Version 1	
*********************************************************************
Version Description:
- initial version
*********************************************************************
Version 2	
*********************************************************************
Version Description:
- Timeout control removed
- Assigning zero when It is not enabled, is removed.
*********************************************************************
*)


IF (C_Enable) THEN						(*Check if the functions is enabled*)
	fb_message(
	iCAN:= Obj_CAN, 
	iCanId:= X_MsgID, 
	iCanIdExtended:= S_Extended, 
	iTimeoutLimit:= Tm_MsgTmOut, 
	oByteCount=> , 
	oData=> , 
	oNewData=> , 
	oCanTimeout=> S_ER_TmOut, 
	oReceiverId=> , 
	oTooManyReceivers=> );	

	IF fb_message.oNewData THEN
	        
	   X_Byte_0 := fb_message.oData[0] ;
	   X_Byte_1 := fb_message.oData[1] ; 
	   X_Byte_2 := fb_message.oData[2] ; 
	   X_Byte_3 := fb_message.oData[3] ;
	   X_Byte_4 := fb_message.oData[4] ;
	   X_Byte_5 := fb_message.oData[5] ;
	   X_Byte_6 := fb_message.oData[6] ;
	   X_Byte_7 := fb_message.oData[7] ;  
	
	END_IF
	
END_IF


                  
END_FUNCTION_BLOCK

FUNCTION_BLOCK _FB_CanRx_Message_Unpack
  VAR_INPUT
    C_Enable : BOOL := FALSE;  (* Enable message *)
    Obj_CAN : POINTER TO tCan;  (* CAN Object derived from CAN_500_LIB *)
    X_MsgID : UDINT := 0;  (* Message ID *)
    Tm_MsgTmOut : TIME := TIME#500ms;  (* Message time limit *)
    S_Extended : BOOL := FALSE;  (* Message extended bit *)
  END_VAR
  VAR_OUTPUT
    S_ER_TmOut : BOOL;  (* Input data endpoints *)
    S_Bit_0 : BOOL;  (* Input data endpoints *)
    S_Bit_1 : BOOL;  (* Input data endpoints *)
    S_Bit_2 : BOOL;  (* Input data endpoints *)
    S_Bit_3 : BOOL;  (* Input data endpoints *)
    S_Bit_4 : BOOL;  (* Input data endpoints *)
    S_Bit_5 : BOOL;  (* Input data endpoints *)
    S_Bit_6 : BOOL;  (* Input data endpoints *)
    S_Bit_7 : BOOL;  (* Input data endpoints *)
    X_Byte_0 : BYTE;  (* Input data endpoints *)
    S_Bit_8 : BOOL;  (* Input data endpoints *)
    S_Bit_9 : BOOL;  (* Input data endpoints *)
    S_Bit_10 : BOOL;  (* Input data endpoints *)
    S_Bit_11 : BOOL;  (* Input data endpoints *)
    S_Bit_12 : BOOL;  (* Input data endpoints *)
    S_Bit_13 : BOOL;  (* Input data endpoints *)
    S_Bit_14 : BOOL;  (* Input data endpoints *)
    S_Bit_15 : BOOL;  (* Input data endpoints *)
    X_Byte_1 : BYTE;  (* Input data endpoints *)
    X_Word_0 : WORD;  (* Input data endpoints *)
    S_Bit_16 : BOOL;  (* Input data endpoints *)
    S_Bit_17 : BOOL;  (* Input data endpoints *)
    S_Bit_18 : BOOL;  (* Input data endpoints *)
    S_Bit_19 : BOOL;  (* Input data endpoints *)
    S_Bit_20 : BOOL;  (* Input data endpoints *)
    S_Bit_21 : BOOL;  (* Input data endpoints *)
    S_Bit_22 : BOOL;  (* Input data endpoints *)
    S_Bit_23 : BOOL;  (* Input data endpoints *)
    X_Byte_2 : BYTE;  (* Input data endpoints *)
    S_Bit_24 : BOOL;  (* Input data endpoints *)
    S_Bit_25 : BOOL;  (* Input data endpoints *)
    S_Bit_26 : BOOL;  (* Input data endpoints *)
    S_Bit_27 : BOOL;  (* Input data endpoints *)
    S_Bit_28 : BOOL;  (* Input data endpoints *)
    S_Bit_29 : BOOL;  (* Input data endpoints *)
    S_Bit_30 : BOOL;  (* Input data endpoints *)
    S_Bit_31 : BOOL;  (* Input data endpoints *)
    X_Byte_3 : BYTE;  (* Input data endpoints *)
    S_Bit_32 : BOOL;  (* Input data endpoints *)
    S_Bit_33 : BOOL;  (* Input data endpoints *)
    S_Bit_34 : BOOL;  (* Input data endpoints *)
    S_Bit_35 : BOOL;  (* Input data endpoints *)
    S_Bit_36 : BOOL;  (* Input data endpoints *)
    S_Bit_37 : BOOL;  (* Input data endpoints *)
    S_Bit_38 : BOOL;  (* Input data endpoints *)
    S_Bit_39 : BOOL;  (* Input data endpoints *)
    X_Byte_4 : BYTE;  (* Input data endpoints *)
    S_Bit_40 : BOOL;  (* Input data endpoints *)
    S_Bit_41 : BOOL;  (* Input data endpoints *)
    S_Bit_42 : BOOL;  (* Input data endpoints *)
    S_Bit_43 : BOOL;  (* Input data endpoints *)
    S_Bit_44 : BOOL;  (* Input data endpoints *)
    S_Bit_45 : BOOL;  (* Input data endpoints *)
    S_Bit_46 : BOOL;  (* Input data endpoints *)
    S_Bit_47 : BOOL;  (* Input data endpoints *)
    X_Byte_5 : BYTE;  (* Input data endpoints *)
    X_Word_2 : WORD;  (* Input data endpoints *)
    S_Bit_48 : BOOL;  (* Input data endpoints *)
    S_Bit_49 : BOOL;  (* Input data endpoints *)
    S_Bit_50 : BOOL;  (* Input data endpoints *)
    S_Bit_51 : BOOL;  (* Input data endpoints *)
    S_Bit_52 : BOOL;  (* Input data endpoints *)
    S_Bit_53 : BOOL;  (* Input data endpoints *)
    S_Bit_54 : BOOL;  (* Input data endpoints *)
    S_Bit_55 : BOOL;  (* Input data endpoints *)
    X_Byte_6 : BYTE;  (* Input data endpoints *)
    S_Bit_56 : BOOL;  (* Input data endpoints *)
    S_Bit_57 : BOOL;  (* Input data endpoints *)
    S_Bit_58 : BOOL;  (* Input data endpoints *)
    S_Bit_59 : BOOL;  (* Input data endpoints *)
    S_Bit_60 : BOOL;  (* Input data endpoints *)
    S_Bit_61 : BOOL;  (* Input data endpoints *)
    S_Bit_62 : BOOL;  (* Input data endpoints *)
    S_Bit_63 : BOOL;  (* Input data endpoints *)
    X_Byte_7 : BYTE;  (* Input data endpoints *)
  END_VAR
  VAR
    fb_message : CanRx;  (* Library object container *)
    STIMEOUT : BOOL;
  END_VAR

                    (*
**********************************************************************
Bozankaya A.Ş.
**********************************************************************
Name					: _FB_CanRx_Message
POU Type				: FB
Created by 				: E.TURKER , BZK.
Creation Date 			: 09-03-2022
Modifications			: see version description below


FB Description:
This FB handles the RX can messages according to CAN_500_LIB
*********************************************************************

Version 1	
*********************************************************************
Version Description:
- initial version
*********************************************************************
Version 2	
*********************************************************************
Version Description:
- Word and dword transitions are removed
*********************************************************************
*)


IF (C_Enable) THEN				(*Check if the function is enabled*)
	fb_message(
	iCAN:= Obj_CAN, 
	iCanId:= X_MsgID, 
	iCanIdExtended:= S_Extended, 
	iTimeoutLimit:= Tm_MsgTmOut, 
	oByteCount=> , 
	oData=> , 
	oNewData=> , 
	oCanTimeout=> S_ER_TmOut, 
	oReceiverId=> , 
	oTooManyReceivers=> );
	
	
	
	IF fb_message.oNewData THEN			(*Check if the new message is received*)

			X_Byte_0 := fb_message.oData[0] ;
			X_Byte_1 := fb_message.oData[1] ; 
			X_Byte_2 := fb_message.oData[2] ; 
			X_Byte_3 := fb_message.oData[3] ;
			X_Byte_4 := fb_message.oData[4] ;
			X_Byte_5 := fb_message.oData[5] ;
			X_Byte_6 := fb_message.oData[6] ;
			X_Byte_7 := fb_message.oData[7] ;  
			
	END_IF
   
	
	
ELSE	
	
			X_Byte_0 := 0 ;
			X_Byte_1 := 0 ;
			X_Byte_2 := 0 ;
			X_Byte_3 := 0 ;
			X_Byte_4 := 0 ;
			X_Byte_5 := 0 ;
			X_Byte_6 := 0 ;
			X_Byte_7 := 0 ;
			
END_IF

			S_Bit_0  := BYTE_TO_BOOL(X_Byte_0 AND 2#00000001);
			S_Bit_1  := BYTE_TO_BOOL(X_Byte_0 AND 2#00000010);
			S_Bit_2  := BYTE_TO_BOOL(X_Byte_0 AND 2#00000100);
			S_Bit_3  := BYTE_TO_BOOL(X_Byte_0 AND 2#00001000);
			S_Bit_4  := BYTE_TO_BOOL(X_Byte_0 AND 2#00010000);
			S_Bit_5  := BYTE_TO_BOOL(X_Byte_0 AND 2#00100000);
			S_Bit_6  := BYTE_TO_BOOL(X_Byte_0 AND 2#01000000);
			S_Bit_7  := BYTE_TO_BOOL(X_Byte_0 AND 2#10000000);
			S_Bit_8  := BYTE_TO_BOOL(X_Byte_1 AND 2#00000001);
			S_Bit_9  := BYTE_TO_BOOL(X_Byte_1 AND 2#00000010);
			S_Bit_10  := BYTE_TO_BOOL(X_Byte_1 AND 2#00000100);
			S_Bit_11  := BYTE_TO_BOOL(X_Byte_1 AND 2#00001000);
			S_Bit_12  := BYTE_TO_BOOL(X_Byte_1 AND 2#00010000);
			S_Bit_13  := BYTE_TO_BOOL(X_Byte_1 AND 2#00100000);
			S_Bit_14  := BYTE_TO_BOOL(X_Byte_1 AND 2#01000000);
			S_Bit_15  := BYTE_TO_BOOL(X_Byte_1 AND 2#10000000);
			S_Bit_16  := BYTE_TO_BOOL(X_Byte_2 AND 2#00000001);
			S_Bit_17  := BYTE_TO_BOOL(X_Byte_2 AND 2#00000010);
			S_Bit_18  := BYTE_TO_BOOL(X_Byte_2 AND 2#00000100);
			S_Bit_19  := BYTE_TO_BOOL(X_Byte_2 AND 2#00001000);
			S_Bit_20  := BYTE_TO_BOOL(X_Byte_2 AND 2#00010000);
			S_Bit_21  := BYTE_TO_BOOL(X_Byte_2 AND 2#00100000);
			S_Bit_22  := BYTE_TO_BOOL(X_Byte_2 AND 2#01000000);
			S_Bit_23  := BYTE_TO_BOOL(X_Byte_2 AND 2#10000000);
			S_Bit_24  := BYTE_TO_BOOL(X_Byte_3 AND 2#00000001);
			S_Bit_25  := BYTE_TO_BOOL(X_Byte_3 AND 2#00000010);
			S_Bit_26  := BYTE_TO_BOOL(X_Byte_3 AND 2#00000100);
			S_Bit_27  := BYTE_TO_BOOL(X_Byte_3 AND 2#00001000);
			S_Bit_28  := BYTE_TO_BOOL(X_Byte_3 AND 2#00010000);
			S_Bit_29  := BYTE_TO_BOOL(X_Byte_3 AND 2#00100000);
			S_Bit_30  := BYTE_TO_BOOL(X_Byte_3 AND 2#01000000);
			S_Bit_31  := BYTE_TO_BOOL(X_Byte_3 AND 2#10000000);
			S_Bit_32  := BYTE_TO_BOOL(X_Byte_4 AND 2#00000001);
			S_Bit_33  := BYTE_TO_BOOL(X_Byte_4 AND 2#00000010);
			S_Bit_34  := BYTE_TO_BOOL(X_Byte_4 AND 2#00000100);
			S_Bit_35  := BYTE_TO_BOOL(X_Byte_4 AND 2#00001000);
			S_Bit_36  := BYTE_TO_BOOL(X_Byte_4 AND 2#00010000);
			S_Bit_37  := BYTE_TO_BOOL(X_Byte_4 AND 2#00100000);
			S_Bit_38  := BYTE_TO_BOOL(X_Byte_4 AND 2#01000000);
			S_Bit_39  := BYTE_TO_BOOL(X_Byte_4 AND 2#10000000);
			S_Bit_40  := BYTE_TO_BOOL(X_Byte_5 AND 2#00000001);
			S_Bit_41  := BYTE_TO_BOOL(X_Byte_5 AND 2#00000010);
			S_Bit_42  := BYTE_TO_BOOL(X_Byte_5 AND 2#00000100);
			S_Bit_43  := BYTE_TO_BOOL(X_Byte_5 AND 2#00001000);
			S_Bit_44  := BYTE_TO_BOOL(X_Byte_5 AND 2#00010000);
			S_Bit_45  := BYTE_TO_BOOL(X_Byte_5 AND 2#00100000);
			S_Bit_46  := BYTE_TO_BOOL(X_Byte_5 AND 2#01000000);
			S_Bit_47  := BYTE_TO_BOOL(X_Byte_5 AND 2#10000000);
			S_Bit_48  := BYTE_TO_BOOL(X_Byte_6 AND 2#00000001);
			S_Bit_49  := BYTE_TO_BOOL(X_Byte_6 AND 2#00000010);
			S_Bit_50  := BYTE_TO_BOOL(X_Byte_6 AND 2#00000100);
			S_Bit_51  := BYTE_TO_BOOL(X_Byte_6 AND 2#00001000);
			S_Bit_52  := BYTE_TO_BOOL(X_Byte_6 AND 2#00010000);
			S_Bit_53  := BYTE_TO_BOOL(X_Byte_6 AND 2#00100000);
			S_Bit_54  := BYTE_TO_BOOL(X_Byte_6 AND 2#01000000);
			S_Bit_55  := BYTE_TO_BOOL(X_Byte_6 AND 2#10000000);
			S_Bit_56  := BYTE_TO_BOOL(X_Byte_7 AND 2#00000001);
			S_Bit_57  := BYTE_TO_BOOL(X_Byte_7 AND 2#00000010);
			S_Bit_58  := BYTE_TO_BOOL(X_Byte_7 AND 2#00000100);
			S_Bit_59  := BYTE_TO_BOOL(X_Byte_7 AND 2#00001000);
			S_Bit_60  := BYTE_TO_BOOL(X_Byte_7 AND 2#00010000);
			S_Bit_61  := BYTE_TO_BOOL(X_Byte_7 AND 2#00100000);
			S_Bit_62  := BYTE_TO_BOOL(X_Byte_7 AND 2#01000000);
			S_Bit_63  := BYTE_TO_BOOL(X_Byte_7 AND 2#10000000);

                  
END_FUNCTION_BLOCK

FUNCTION_BLOCK _FB_CanTx_Message
  VAR_INPUT
    C_Enable : BOOL := FALSE;  (* Enable message *)
    Obj_CAN : POINTER TO tCan;  (* CAN Object derived from CAN_500_LIB *)
    X_MsgID : UDINT := 0;  (* Message ID *)
    Tm_CycleTime : TIME := TIME#500ms;  (* Message time limit *)
    N_Msg_Dlc : BYTE := 8;  (* Message dlc *)
    S_Extended : BOOL := FALSE;  (* Message extended bit *)
    X_Byte_0 : BYTE := 16#FF;  (* Message Datas *)
    X_Byte_1 : BYTE := 16#FF;  (* Message Datas *)
    X_Byte_2 : BYTE := 16#FF;  (* Message Datas *)
    X_Byte_3 : BYTE := 16#FF;  (* Message Datas *)
    X_Byte_4 : BYTE := 16#FF;  (* Message Datas *)
    X_Byte_5 : BYTE := 16#FF;  (* Message Datas *)
    X_Byte_6 : BYTE := 16#FF;  (* Message Datas *)
    X_Byte_7 : BYTE := 16#FF;  (* Message Datas *)
  END_VAR
  VAR_OUTPUT
    S_Sent_Ok : BOOL;  (* Data sent acknowledge *)
  END_VAR
  VAR
    fb_message : CanTx;  (* Library object container *)
    Arr_X_Data : ARRAY[0..7] OF BYTE;  (* Message data array *)
  END_VAR

                    (*
**********************************************************************
Bozankaya A.Ş.
**********************************************************************
Name					: _FB_CanTx_Message
POU Type				: FB
Created by 				: E.TURKER , BZK.
Creation Date 			: 09-03-2022
Modifications			: see version description below


FB Description:
This FB handles the TX can messages according to CAN_500_LIB
*********************************************************************

Version 1	
*********************************************************************
Version Description:
- initial version
*********************************************************************
Version 2	
*********************************************************************
Version Description:
- Assigning zero when It is not enabled, is removed.
*********************************************************************
*)

IF C_Enable THEN				(*Check if the function is enabled*)
			
			Arr_X_Data [0] := X_Byte_0;
			Arr_X_Data [1] := X_Byte_1;
			Arr_X_Data [2] := X_Byte_2;
			Arr_X_Data [3] := X_Byte_3;
			Arr_X_Data [4] := X_Byte_4;
			Arr_X_Data [5] := X_Byte_5;		
            Arr_X_Data [6] := X_Byte_6;
			Arr_X_Data [7] := X_Byte_7;

END_IF

fb_message(
	
	iEnable:= C_Enable, 
	iCAN:= Obj_CAN, 
	iForceSend:= FALSE, 
	iTransmitRate:= Tm_CycleTime, 
	iCanId:= X_MsgID, 
	iCanIdExtended:= S_Extended, 
	iByteCount:= N_Msg_Dlc, 
	iData:= Arr_X_Data, 
	oTransmitterId=> , 
	oTooManyTransmitters=> , 
	oMsgSent=> S_Sent_Ok );
	
                  
END_FUNCTION_BLOCK

FUNCTION_BLOCK _FB_CanTx_Message_Unpack
  VAR_INPUT
    C_Enable : BOOL := FALSE;  (* Enable message *)
    Obj_CAN : POINTER TO tCan;  (* CAN Object derived from CAN_500_LIB *)
    X_MsgID : UDINT := 0;  (* Message ID *)
    Tm_CycleTime : TIME := TIME#500ms;  (* Message time limit *)
    S_Extended : BOOL := FALSE;  (* Message extended bit *)
    N_Msg_Dlc : BYTE;
    S_Bit_0 : BOOL := FALSE;  (* Message Datas *)
    S_Bit_1 : BOOL := FALSE;  (* Message Datas *)
    S_Bit_2 : BOOL := FALSE;  (* Message Datas *)
    S_Bit_3 : BOOL := FALSE;  (* Message Datas *)
    S_Bit_4 : BOOL := FALSE;  (* Message Datas *)
    S_Bit_5 : BOOL := FALSE;  (* Message Datas *)
    S_Bit_6 : BOOL := FALSE;  (* Message Datas *)
    S_Bit_7 : BOOL := FALSE;  (* Message Datas *)
    X_Byte_0 : BYTE := 16#0;  (* Message Datas *)
    S_Bit_8 : BOOL := FALSE;  (* Message Datas *)
    S_Bit_9 : BOOL := FALSE;  (* Message Datas *)
    S_Bit_10 : BOOL := FALSE;  (* Message Datas *)
    S_Bit_11 : BOOL := FALSE;  (* Message Datas *)
    S_Bit_12 : BOOL := FALSE;  (* Message Datas *)
    S_Bit_13 : BOOL := FALSE;  (* Message Datas *)
    S_Bit_14 : BOOL := FALSE;  (* Message Datas *)
    S_Bit_15 : BOOL := FALSE;  (* Message Datas *)
    X_Byte_1 : BYTE := 16#0;  (* Message Datas *)
    S_Bit_16 : BOOL := FALSE;  (* Message Datas *)
    S_Bit_17 : BOOL := FALSE;  (* Message Datas *)
    S_Bit_18 : BOOL := FALSE;  (* Message Datas *)
    S_Bit_19 : BOOL := FALSE;  (* Message Datas *)
    S_Bit_20 : BOOL := FALSE;  (* Message Datas *)
    S_Bit_21 : BOOL := FALSE;  (* Message Datas *)
    S_Bit_22 : BOOL := FALSE;  (* Message Datas *)
    S_Bit_23 : BOOL := FALSE;  (* Message Datas *)
    X_Byte_2 : BYTE := 16#0;  (* Message Datas *)
    S_Bit_24 : BOOL := FALSE;  (* Message Datas *)
    S_Bit_25 : BOOL := FALSE;  (* Message Datas *)
    S_Bit_26 : BOOL := FALSE;  (* Message Datas *)
    S_Bit_27 : BOOL := FALSE;  (* Message Datas *)
    S_Bit_28 : BOOL := FALSE;  (* Message Datas *)
    S_Bit_29 : BOOL := FALSE;  (* Message Datas *)
    S_Bit_30 : BOOL := FALSE;  (* Message Datas *)
    S_Bit_31 : BOOL := FALSE;  (* Message Datas *)
    X_Byte_3 : BYTE := 16#0;  (* Message Datas *)
    S_Bit_32 : BOOL := FALSE;  (* Message Datas *)
    S_Bit_33 : BOOL := FALSE;  (* Message Datas *)
    S_Bit_34 : BOOL := FALSE;  (* Message Datas *)
    S_Bit_35 : BOOL := FALSE;  (* Message Datas *)
    S_Bit_36 : BOOL := FALSE;  (* Message Datas *)
    S_Bit_37 : BOOL := FALSE;  (* Message Datas *)
    S_Bit_38 : BOOL := FALSE;  (* Message Datas *)
    S_Bit_39 : BOOL := FALSE;  (* Message Datas *)
    X_Byte_4 : BYTE := 16#0;  (* Message Datas *)
    S_Bit_40 : BOOL := FALSE;  (* Message Datas *)
    S_Bit_41 : BOOL := FALSE;  (* Message Datas *)
    S_Bit_42 : BOOL := FALSE;  (* Message Datas *)
    S_Bit_43 : BOOL := FALSE;  (* Message Datas *)
    S_Bit_44 : BOOL := FALSE;  (* Message Datas *)
    S_Bit_45 : BOOL := FALSE;  (* Message Datas *)
    S_Bit_46 : BOOL := FALSE;  (* Message Datas *)
    S_Bit_47 : BOOL := FALSE;  (* Message Datas *)
    X_Byte_5 : BYTE := 16#0;  (* Message Datas *)
    S_Bit_48 : BOOL := FALSE;  (* Message Datas *)
    S_Bit_49 : BOOL := FALSE;  (* Message Datas *)
    S_Bit_50 : BOOL := FALSE;  (* Message Datas *)
    S_Bit_51 : BOOL := FALSE;  (* Message Datas *)
    S_Bit_52 : BOOL := FALSE;  (* Message Datas *)
    S_Bit_53 : BOOL := FALSE;  (* Message Datas *)
    S_Bit_54 : BOOL := FALSE;  (* Message Datas *)
    S_Bit_55 : BOOL := FALSE;  (* Message Datas *)
    X_Byte_6 : BYTE := 16#0;  (* Message Datas *)
    S_Bit_56 : BOOL := FALSE;  (* Message Datas *)
    S_Bit_57 : BOOL := FALSE;  (* Message Datas *)
    S_Bit_58 : BOOL := FALSE;  (* Message Datas *)
    S_Bit_59 : BOOL := FALSE;  (* Message Datas *)
    S_Bit_60 : BOOL := FALSE;  (* Message Datas *)
    S_Bit_61 : BOOL := FALSE;  (* Message Datas *)
    S_Bit_62 : BOOL := FALSE;  (* Message Datas *)
    S_Bit_63 : BOOL := FALSE;  (* Message Datas *)
    X_Byte_7 : BYTE := 16#0;  (* Message Datas *)
  END_VAR
  VAR_OUTPUT
    S_Sent_Ok : BOOL;  (* Data sent acknowledge *)
  END_VAR
  VAR
    fb_message : CanTx;  (* Library object container *)
    DATA : ARRAY[0..7] OF BYTE;  (* Message data array *)
    _FB_Pack_Bit_To_Byte_01 : _FB_PACK_8BITS_TO_BYTE;
    _FB_Pack_Bit_To_Byte_02 : _FB_PACK_8BITS_TO_BYTE;
    _FB_Pack_Bit_To_Byte_03 : _FB_PACK_8BITS_TO_BYTE;
    _FB_Pack_Bit_To_Byte_04 : _FB_PACK_8BITS_TO_BYTE;
    _FB_Pack_Bit_To_Byte_05 : _FB_PACK_8BITS_TO_BYTE;
    _FB_Pack_Bit_To_Byte_06 : _FB_PACK_8BITS_TO_BYTE;
    _FB_Pack_Bit_To_Byte_07 : _FB_PACK_8BITS_TO_BYTE;
    _FB_Pack_Bit_To_Byte_08 : _FB_PACK_8BITS_TO_BYTE;
  END_VAR

                    (*
**********************************************************************
Bozankaya A.Ş.
**********************************************************************
Name					: _FB_CanTx_Message
POU Type				: FB
Created by 				: E.TURKER , BZK.
Creation Date 			: 09-03-2022
Modifications			: see version description below


FB Description:
This FB handles the TX can messages according to CAN_500_LIB
*********************************************************************

Version 1	
*********************************************************************
Version Description:
- initial version
*********************************************************************
Version 1	
*********************************************************************
Version Description:
- WORD and DWORD transitions are removed
*********************************************************************
*)

IF X_Byte_0 <> 0 THEN
	
	DATA [0] := X_Byte_0;
	
ELSIF S_Bit_0 OR S_Bit_1 OR S_Bit_2 OR S_Bit_3 OR S_Bit_4 OR S_Bit_5 OR S_Bit_6 OR S_Bit_7 THEN			(*Check the bits, pack and assign to the output data*)
	_FB_Pack_Bit_To_Byte_01(
	S_Bit_0:= S_Bit_0, 
	S_Bit_1:= S_Bit_1, 
	S_Bit_2:= S_Bit_2, 
	S_Bit_3:= S_Bit_3, 
	S_Bit_4:= S_Bit_4, 
	S_Bit_5:= S_Bit_5, 
	S_Bit_6:= S_Bit_6, 
	S_Bit_7:= S_Bit_7, 
	X_Byte_0=> DATA [0]);
ELSE
	DATA [0] := 0;
END_IF
		
IF X_Byte_1 <> 0 THEN
	DATA [1] := X_Byte_1;
ELSIF S_Bit_8 OR S_Bit_9 OR S_Bit_10 OR S_Bit_11 OR S_Bit_12 OR S_Bit_13 OR S_Bit_14 OR S_Bit_15 THEN			(*Check the bits, pack and assign to the output data*)
	_FB_Pack_Bit_To_Byte_02(
	S_Bit_0:= S_Bit_8, 
	S_Bit_1:= S_Bit_9, 
	S_Bit_2:= S_Bit_10, 
	S_Bit_3:= S_Bit_11, 
	S_Bit_4:= S_Bit_12, 
	S_Bit_5:= S_Bit_13, 
	S_Bit_6:= S_Bit_14, 
	S_Bit_7:= S_Bit_15, 
	X_Byte_0=> DATA [1]);
ELSE
	DATA [1] :=0;
END_IF
	

IF X_Byte_2 <> 0 THEN
	DATA [2] := X_Byte_2;
ELSIF S_Bit_16 OR S_Bit_17 OR S_Bit_18 OR S_Bit_19 OR S_Bit_20 OR S_Bit_21 OR S_Bit_22 OR S_Bit_23 THEN				(*Check the bits, pack and assign to the output data*)
	_FB_Pack_Bit_To_Byte_03(
	S_Bit_0:= S_Bit_16, 
	S_Bit_1:= S_Bit_17, 
	S_Bit_2:= S_Bit_18, 
	S_Bit_3:= S_Bit_19, 
	S_Bit_4:= S_Bit_20, 
	S_Bit_5:= S_Bit_21, 
	S_Bit_6:= S_Bit_22, 
	S_Bit_7:= S_Bit_23, 
	X_Byte_0=> DATA [2]);
ELSE
	DATA [2] :=0;
END_IF
		
IF X_Byte_3 <> 0 THEN
	DATA [3] := X_Byte_3;
ELSIF S_Bit_24 OR S_Bit_25 OR S_Bit_26 OR S_Bit_27 OR S_Bit_28 OR S_Bit_29 OR S_Bit_30 OR S_Bit_31 THEN				(*Check the bits, pack and assign to the output data*)
	_FB_Pack_Bit_To_Byte_04(
	S_Bit_0:= S_Bit_24, 
	S_Bit_1:= S_Bit_25, 
	S_Bit_2:= S_Bit_26, 
	S_Bit_3:= S_Bit_27, 
	S_Bit_4:= S_Bit_28, 
	S_Bit_5:= S_Bit_29, 
	S_Bit_6:= S_Bit_30, 
	S_Bit_7:= S_Bit_31, 
	X_Byte_0=> DATA [3]);
ELSE
	DATA [3] :=0;
END_IF



IF X_Byte_4 <> 0 THEN
	DATA [4] := X_Byte_4;
ELSIF S_Bit_32 OR S_Bit_33 OR S_Bit_34 OR S_Bit_35 OR S_Bit_36 OR S_Bit_37 OR S_Bit_38 OR S_Bit_39 THEN				(*Check the bits, pack and assign to the output data*)
	_FB_Pack_Bit_To_Byte_05(
	S_Bit_0:= S_Bit_32, 
	S_Bit_1:= S_Bit_33, 
	S_Bit_2:= S_Bit_34, 
	S_Bit_3:= S_Bit_35, 
	S_Bit_4:= S_Bit_36, 
	S_Bit_5:= S_Bit_37, 
	S_Bit_6:= S_Bit_38, 
	S_Bit_7:= S_Bit_39, 
	X_Byte_0=> DATA [4]);	
ELSE
	DATA [4] :=0;
END_IF
		
IF X_Byte_5 <> 0 THEN
	DATA [5] := X_Byte_5;
ELSIF S_Bit_40 OR S_Bit_41 OR S_Bit_42 OR S_Bit_43 OR S_Bit_44 OR S_Bit_45 OR S_Bit_46 OR S_Bit_47 THEN				(*Check the bits, pack and assign to the output data*)
	_FB_Pack_Bit_To_Byte_06(
	S_Bit_0:= S_Bit_40, 
	S_Bit_1:= S_Bit_41, 
	S_Bit_2:= S_Bit_42, 
	S_Bit_3:= S_Bit_43, 
	S_Bit_4:= S_Bit_44, 
	S_Bit_5:= S_Bit_45, 
	S_Bit_6:= S_Bit_46, 
	S_Bit_7:= S_Bit_47, 
	X_Byte_0=> DATA [5]);
ELSE
	DATA [5] :=0;
END_IF

	

IF X_Byte_6 <> 0 THEN
	DATA [6] := X_Byte_6;
ELSIF S_Bit_48 OR S_Bit_49 OR S_Bit_50 OR S_Bit_51 OR S_Bit_52 OR S_Bit_53 OR S_Bit_54 OR S_Bit_55 THEN				(*Check the bits, pack and assign to the output data*)
	_FB_Pack_Bit_To_Byte_07(
	S_Bit_0:= S_Bit_48, 
	S_Bit_1:= S_Bit_49, 
	S_Bit_2:= S_Bit_50, 
	S_Bit_3:= S_Bit_51, 
	S_Bit_4:= S_Bit_52, 
	S_Bit_5:= S_Bit_53, 
	S_Bit_6:= S_Bit_54, 
	S_Bit_7:= S_Bit_55, 
	X_Byte_0=> DATA [6]);
ELSE
	DATA [6] :=0;
END_IF
		
IF X_Byte_7 <> 0 THEN
	DATA [7] := X_Byte_7;
ELSIF S_Bit_56 OR S_Bit_57 OR S_Bit_58 OR S_Bit_59 OR S_Bit_60 OR S_Bit_61 OR S_Bit_62 OR S_Bit_63 THEN				(*Check the bits, pack and assign to the output data*)
	_FB_Pack_Bit_To_Byte_08(
	S_Bit_0:= S_Bit_56, 
	S_Bit_1:= S_Bit_57, 
	S_Bit_2:= S_Bit_58, 
	S_Bit_3:= S_Bit_59, 
	S_Bit_4:= S_Bit_60, 
	S_Bit_5:= S_Bit_61, 
	S_Bit_6:= S_Bit_62, 
	S_Bit_7:= S_Bit_63, 
	X_Byte_0=> DATA [7]);
ELSE
	DATA [7] :=0;
END_IF


fb_message(
	iEnable:= C_Enable, 
	iCAN:= Obj_CAN, 
	iForceSend:= FALSE, 
	iTransmitRate:= Tm_CycleTime, 
	iCanId:= X_MsgID, 
	iCanIdExtended:= S_Extended, 
	iByteCount:= N_Msg_Dlc, 
	iData:= DATA, 
	oTransmitterId=> , 
	oTooManyTransmitters=> , 
	oMsgSent=> S_Sent_Ok );
                  
END_FUNCTION_BLOCK

FUNCTION_BLOCK _FB_LfMon
  VAR_INPUT
    X_Lf : UINT;
    P_Lf_Timeout : TIME;
  END_VAR
  VAR_OUTPUT
    S_Lf_Timeout : BOOL;
  END_VAR
  VAR
    X_Lf_Old : UINT;
    TON_0 : TON;
  END_VAR

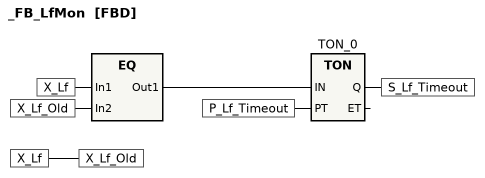
(* FBD diagram, written out as Structured Text *)
TON_0(IN := X_Lf = X_Lf_Old, PT := P_Lf_Timeout);
S_Lf_Timeout := TON_0.Q;
X_Lf_Old := X_Lf;
END_FUNCTION_BLOCK

FUNCTION_BLOCK _FB_PACK_8BITS_TO_BYTE
  VAR_INPUT
    S_BIT_0 : BOOL;  (* Less significant part *)
    S_BIT_1 : BOOL;
    S_BIT_2 : BOOL;
    S_BIT_3 : BOOL;
    S_BIT_4 : BOOL;
    S_BIT_5 : BOOL;
    S_BIT_6 : BOOL;
    S_BIT_7 : BOOL;  (* Most significant part *)
  END_VAR
  VAR_OUTPUT
    X_BYTE_0 : BYTE;  (* Output data *)
  END_VAR
  VAR
    X_Cont_Byte : BYTE;  (* Container data for shifting operation *)
  END_VAR

                    X_Cont_Byte 	:= BOOL_TO_BYTE(S_BIT_7) OR X_Cont_Byte;			
X_Cont_Byte		:= SHL(X_Cont_Byte, 1);
X_Cont_Byte     := BOOL_TO_BYTE(S_BIT_6) OR X_Cont_Byte;
X_Cont_Byte		:= SHL(X_Cont_Byte, 1);
X_Cont_Byte     := BOOL_TO_BYTE(S_BIT_5) OR X_Cont_Byte;
X_Cont_Byte		:= SHL(X_Cont_Byte, 1);
X_Cont_Byte     := BOOL_TO_BYTE(S_BIT_4) OR X_Cont_Byte;
X_Cont_Byte		:= SHL(X_Cont_Byte, 1);
X_Cont_Byte     := BOOL_TO_BYTE(S_BIT_3) OR X_Cont_Byte;
X_Cont_Byte		:= SHL(X_Cont_Byte, 1);
X_Cont_Byte     := BOOL_TO_BYTE(S_BIT_2) OR X_Cont_Byte;
X_Cont_Byte		:= SHL(X_Cont_Byte, 1);
X_Cont_Byte     := BOOL_TO_BYTE(S_BIT_1) OR X_Cont_Byte;
X_Cont_Byte		:= SHL(X_Cont_Byte, 1);
X_Cont_Byte     := BOOL_TO_BYTE(S_BIT_0) OR X_Cont_Byte;
X_BYTE_0		:= X_Cont_Byte;
X_Cont_Byte		:=0;
                  
END_FUNCTION_BLOCK

FUNCTION_BLOCK _FB_PACK_BYTE_TO_DINT
  VAR_INPUT
    X_Byte_0 : BYTE;  (* Input less significant part *)
    X_Byte_1 : BYTE;
    X_Byte_2 : BYTE;
    X_Byte_3 : BYTE;
    X_Byte_4 : BYTE;
    X_Byte_5 : BYTE;
    X_Byte_6 : BYTE;
    X_Byte_7 : BYTE;  (* Input most significant part *)
  END_VAR
  VAR_OUTPUT
    X_Dint_0 : DINT;
  END_VAR
  VAR
    X_Cont_Udint : UDINT;  (* Container data for shifting operation *)
  END_VAR

                    X_Cont_Udint	:= BYTE_TO_UDINT(X_Byte_3) OR X_Cont_Udint;
X_Cont_Udint	:= SHL(X_Cont_Udint, 8);
X_Cont_Udint	:= BYTE_TO_UDINT(X_Byte_2) OR X_Cont_Udint;
X_Cont_Udint	:= SHL(X_Cont_Udint, 8);
X_Cont_Udint	:= BYTE_TO_UDINT(X_Byte_1) OR X_Cont_Udint;
X_Cont_Udint	:= SHL(X_Cont_Udint, 8);
X_Cont_Udint	:= BYTE_TO_UDINT(X_Byte_0) OR X_Cont_Udint;
X_Dint_0 := UDINT_TO_DINT(X_Cont_Udint);
X_Cont_Udint:=0;
                  
END_FUNCTION_BLOCK

FUNCTION_BLOCK _FB_PACK_BYTE_TO_DWORD
  VAR_INPUT
    X_BYTE_0 : BYTE;  (* Input less significant part *)
    X_BYTE_1 : BYTE;  (* Input most significant part *)
    X_BYTE_2 : BYTE;  (* Input less significant part *)
    X_BYTE_3 : BYTE;  (* Input most significant part *)
  END_VAR
  VAR_OUTPUT
    X_DWORD_0 : DWORD;  (* Output data *)
  END_VAR
  VAR
    X_Cont_DWord : DWORD;  (* Container data for shifting operation *)
  END_VAR

                    X_Cont_DWord 	:= BYTE_TO_DWORD(X_BYTE_3) OR X_Cont_DWord;			
X_Cont_DWord	:= SHL(X_Cont_DWord, 8);
X_Cont_DWord    := BYTE_TO_DWORD(X_BYTE_2) OR X_Cont_DWord;
X_Cont_DWord	:= SHL(X_Cont_DWord, 8);
X_Cont_DWord    := BYTE_TO_DWORD(X_BYTE_1) OR X_Cont_DWord;
X_Cont_DWord	:= SHL(X_Cont_DWord, 8);
X_Cont_DWord    := BYTE_TO_DWORD(X_BYTE_0) OR X_Cont_DWord;
X_DWORD_0		:= X_Cont_DWord;
X_Cont_DWord	:= 0;
                  
END_FUNCTION_BLOCK

FUNCTION_BLOCK _FB_PACK_BYTE_TO_INT
  VAR_INPUT
    X_Byte_0 : BYTE;  (* Input less significant part *)
    X_Byte_1 : BYTE;  (* Input most significant part *)
  END_VAR
  VAR_OUTPUT
    X_Int_0 : INT;
  END_VAR
  VAR
    X_Cont_Uint : UINT;  (* Container data for shifting operation *)
  END_VAR

                    X_Cont_Uint 	:= BYTE_TO_UINT(X_Byte_1) OR X_Cont_Uint;
X_Cont_Uint		:= SHL(X_Cont_Uint, 8);
X_Cont_Uint		:= BYTE_TO_UINT(X_Byte_0) OR X_Cont_Uint;
X_Int_0   		:= UINT_TO_INT(X_Cont_Uint);
X_Cont_Uint:=0;
                  
END_FUNCTION_BLOCK

FUNCTION_BLOCK _FB_PACK_BYTE_TO_LWORD
  VAR_INPUT
    X_BYTE_0 : BYTE;  (* Input less significant part *)
    X_BYTE_1 : BYTE;  (* Input most significant part *)
    X_BYTE_2 : BYTE;  (* Input less significant part *)
    X_BYTE_3 : BYTE;  (* Input most significant part *)
    X_BYTE_4 : BYTE;  (* Input less significant part *)
    X_BYTE_5 : BYTE;  (* Input most significant part *)
    X_BYTE_6 : BYTE;  (* Input less significant part *)
    X_BYTE_7 : BYTE;  (* Input most significant part *)
  END_VAR
  VAR_OUTPUT
    X_LWORD_0 : LWORD;  (* Output data *)
  END_VAR
  VAR
    X_Cont_LWord : LWORD;  (* Container data for shifting operation *)
  END_VAR

                    X_Cont_LWord 	:= BYTE_TO_LWORD(X_BYTE_7) OR X_Cont_LWord;			
X_Cont_LWord	:= SHL(X_Cont_LWord, 8);
X_Cont_LWord    := BYTE_TO_LWORD(X_BYTE_6) OR X_Cont_LWord;
X_Cont_LWord	:= SHL(X_Cont_LWord, 8);
X_Cont_LWord    := BYTE_TO_LWORD(X_BYTE_5) OR X_Cont_LWord;
X_Cont_LWord	:= SHL(X_Cont_LWord, 8);
X_Cont_LWord    := BYTE_TO_LWORD(X_BYTE_4) OR X_Cont_LWord;
X_Cont_LWord	:= SHL(X_Cont_LWord, 8);
X_Cont_LWord    := BYTE_TO_LWORD(X_BYTE_3) OR X_Cont_LWord;
X_Cont_LWord	:= SHL(X_Cont_LWord, 8);
X_Cont_LWord    := BYTE_TO_LWORD(X_BYTE_2) OR X_Cont_LWord;
X_Cont_LWord	:= SHL(X_Cont_LWord, 8);
X_Cont_LWord    := BYTE_TO_LWORD(X_BYTE_1) OR X_Cont_LWord;
X_Cont_LWord	:= SHL(X_Cont_LWord, 8);
X_Cont_LWord    := BYTE_TO_LWORD(X_BYTE_0) OR X_Cont_LWord;
X_LWORD_0		:= X_Cont_LWord;
X_Cont_LWord	:= 0;
                  
END_FUNCTION_BLOCK

FUNCTION_BLOCK _FB_PACK_BYTE_TO_UINT
  VAR_INPUT
    X_BYTE_0 : BYTE;  (* Input less significant part *)
    X_BYTE_1 : BYTE;  (* Input most significant part *)
  END_VAR
  VAR_OUTPUT
    X_UINT_0 : UINT;  (* Output Data *)
  END_VAR
  VAR
    X_Cont_Uint : UINT;  (* Container data for shifting operation *)
  END_VAR

                    X_Cont_Uint := 	BYTE_TO_UINT(X_BYTE_1) OR X_Cont_Uint;
X_Cont_Uint	:= 	SHL(X_Cont_Uint, 8);
X_Cont_Uint := 	BYTE_TO_UINT(X_BYTE_0) OR X_Cont_Uint;
X_UINT_0	:=	X_Cont_Uint ;
X_Cont_Uint	:=	0;
                  
END_FUNCTION_BLOCK

FUNCTION_BLOCK _FB_PACK_BYTE_TO_ULINT
  VAR_INPUT
    X_BYTE_0 : BYTE;  (* Input less significant part *)
    X_BYTE_1 : BYTE;
    X_BYTE_2 : BYTE;
    X_BYTE_3 : BYTE;
    X_BYTE_4 : BYTE;
    X_BYTE_5 : BYTE;
    X_BYTE_6 : BYTE;
    X_BYTE_7 : BYTE;  (* Input most significant part *)
  END_VAR
  VAR_OUTPUT
    X_ULINT_0 : ULINT;  (* Output data *)
  END_VAR
  VAR
    X_Cont_Ulint : ULINT;  (* Container data for shifting operation *)
  END_VAR

                    X_Cont_Ulint	:= BYTE_TO_USINT(X_BYTE_7) OR X_Cont_Ulint;
X_Cont_Ulint	:= SHL(X_Cont_Ulint, 8);
X_Cont_Ulint	:= BYTE_TO_USINT(X_BYTE_6) OR X_Cont_Ulint;
X_Cont_Ulint	:= SHL(X_Cont_Ulint, 8);
X_Cont_Ulint	:= BYTE_TO_USINT(X_BYTE_5) OR X_Cont_Ulint;
X_Cont_Ulint	:= SHL(X_Cont_Ulint, 8);
X_Cont_Ulint	:= BYTE_TO_USINT(X_BYTE_4) OR X_Cont_Ulint;
X_Cont_Ulint	:= SHL(X_Cont_Ulint, 8);
X_Cont_Ulint	:= BYTE_TO_USINT(X_BYTE_3) OR X_Cont_Ulint;
X_Cont_Ulint	:= SHL(X_Cont_Ulint, 8);
X_Cont_Ulint	:= BYTE_TO_USINT(X_BYTE_2) OR X_Cont_Ulint;
X_Cont_Ulint	:= SHL(X_Cont_Ulint, 8);
X_Cont_Ulint	:= BYTE_TO_USINT(X_BYTE_1) OR X_Cont_Ulint;
X_Cont_Ulint	:= SHL(X_Cont_Ulint, 8);
X_Cont_Ulint	:= BYTE_TO_USINT(X_BYTE_0) OR X_Cont_Ulint;
X_ULINT_0 		:= X_Cont_Ulint;
X_Cont_Ulint	:=	0;
                  
END_FUNCTION_BLOCK

FUNCTION_BLOCK _FB_PACK_BYTE_TO_WORD
  VAR_INPUT
    X_BYTE_0 : BYTE;  (* Input less significant part *)
    X_BYTE_1 : BYTE;  (* Input most significant part *)
  END_VAR
  VAR_OUTPUT
    X_WORD_0 : WORD;  (* Output data *)
  END_VAR
  VAR
    X_Cont_Word : WORD;  (* Container data for shifting operation *)
  END_VAR

                    X_Cont_Word 	:= BYTE_TO_WORD(X_BYTE_1) OR X_Cont_Word;			
X_Cont_Word		:= SHL(X_Cont_Word, 8);
X_Cont_Word     := BYTE_TO_WORD(X_BYTE_0) OR X_Cont_Word;
X_WORD_0		:= X_Cont_Word;
X_Cont_Word		:=0;
                  
END_FUNCTION_BLOCK

FUNCTION_BLOCK _FB_PACK_DWORD_TO_LWORD
  VAR_INPUT
    X_DWORD_0 : DWORD;  (* Input less significant part *)
    X_DWORD_1 : DWORD;  (* Input most significant part *)
  END_VAR
  VAR_OUTPUT
    X_LWORD_0 : LWORD;  (* Output data *)
  END_VAR
  VAR
    X_Cont_LWord : LWORD;  (* Container data for shifting operation *)
  END_VAR

                    X_Cont_LWord 	:= DWORD_TO_LWORD(X_DWORD_1) OR X_Cont_LWord;			
X_Cont_LWord	:= SHL(X_Cont_LWord, 16);
X_Cont_LWord    := DWORD_TO_LWORD(X_DWORD_0) OR X_Cont_LWord;
X_LWORD_0		:= X_Cont_LWord;
X_Cont_LWord	:= 0;
                  
END_FUNCTION_BLOCK

FUNCTION_BLOCK _FB_PACK_WORD_TO_DWORD
  VAR_INPUT
    X_WORD_0 : WORD;  (* Input less significant part *)
    X_WORD_1 : WORD;  (* Input most significant part *)
  END_VAR
  VAR_OUTPUT
    X_DWORD_0 : DWORD;  (* Output data *)
  END_VAR
  VAR
    X_Cont_DWord : DWORD;  (* Container data for shifting operation *)
  END_VAR

                    X_Cont_DWord 	:= WORD_TO_DWORD(X_WORD_1) OR X_Cont_DWord;			
X_Cont_DWord	:= SHL(X_Cont_DWord, 16);
X_Cont_DWord    := WORD_TO_DWORD(X_WORD_0) OR X_Cont_DWord;
X_DWORD_0		:= X_Cont_DWord;
X_Cont_DWord	:= 0;
                  
END_FUNCTION_BLOCK

FUNCTION_BLOCK _FB_Selector_
  VAR_INPUT
    I1_Value : REAL;
    I1_Valid : BOOL;
    I2_Value : REAL;
    I2_Valid : BOOL;
    I3_Value : REAL;
    I3_Valid : BOOL;
  END_VAR
  VAR_OUTPUT
    O_Value : REAL;
  END_VAR

                    IF I1_Valid THEN
	O_Value:=I1_Value;
ELSIF I2_Valid THEN
	O_Value:=I2_Value;
ELSIF I3_Valid THEN
	O_Value:=I3_Value;
END_IF
                  
END_FUNCTION_BLOCK

FUNCTION_BLOCK _FB_Stm_4Node
  VAR_INPUT
    S_Trans_S0S10 : BOOL := FALSE;  (* Transitions from IDLE TO State 10 *)
    S_Trans_S10S20 : BOOL := FALSE;  (* Transitions from State 10 TO State 20 *)
    S_Trans_S10S30 : BOOL := FALSE;
    S_Trans_S10S40 : BOOL := FALSE;
    Tm_TmOut_S10 : TIME := TIME#28800m0s0ms;
    S_Trans_S20S10 : BOOL := FALSE;  (* Transitions from State 20 TO Other states *)
    S_Trans_S20S30 : BOOL := FALSE;
    S_Trans_S20S40 : BOOL := FALSE;
    Tm_TmOut_S20 : TIME := TIME#28800m0s0ms;
    S_Trans_S30S10 : BOOL := FALSE;  (* Transitions from State 30 TO Other states *)
    S_Trans_S30S20 : BOOL := FALSE;
    S_Trans_S30S40 : BOOL := FALSE;
    Tm_TmOut_S30 : TIME := TIME#28800m0s0ms;
    S_Trans_S40S10 : BOOL := FALSE;  (* Transition from State 40 TO Other states *)
    S_Trans_S40S20 : BOOL := FALSE;
    S_Trans_S40S30 : BOOL := FALSE;
    Tm_TmOut_S40 : TIME := TIME#28800m0s0ms;
    Tm_Sys : TIME;  (* System RTC Time *)
  END_VAR
  VAR_OUTPUT
    S_Idle : BOOL;
    S_Stat10 : BOOL;
    S_Stat20 : BOOL;
    S_Stat30 : BOOL;
    S_Stat40 : BOOL;
  END_VAR
  VAR
    POU_Version : WSTRING;
    X_Act_Old : UINT := 0;  (* Old state node *)
    X_Act_St : UINT := 0;  (* Active state node *)
    S_New_Node : BOOL := TRUE;  (* Old node and actual node is different at the end of state *)
    Tm_Node_Entry : TIME := TIME#0ms;  (* Node entry time *)
    Tm_Actual : TIME := TIME#0ms;  (* Actual time *)
    _FB_Tools_Shf_RegStm_01 : _FB_Tools_Shf_RegStm;  (* Shift register to monitor last 8 state *)
    XActStat : INT;  (* _FUN_Tools_TmOutStm_01 : _FUN_Tools_TmOutStm ; ( *Timout control function depending to actual and node entry time* ) *)
  END_VAR

                    (*
**********************************************************************
Bozankaya A.Ş.
**********************************************************************
Name					: _FB_Stm_4Node
POU Type				: FB
Created by 				: E.TURKER , BZK.
Creation Date 			: 17-03-2022
Modifications			: see version description below


FB Description:
This FB handles the basic integrity of state machines. 
Features:
		Stores last 8 node state
		Checks timeout state on every node
		
--------------Do not edit on application usage purpose.---------------
*********************************************************************

Version 1	
*********************************************************************
Version Description:
- initial version
*********************************************************************
*)




POU_Version := "V0.1";


IF S_New_Node THEN
	Tm_Node_Entry := Tm_Sys;		(*Assign system time when the new entry detected*)
END_IF;
X_Act_Old := X_Act_St;			
Tm_Actual := Tm_Sys;		(*Assign system to actual time register on every cycle*)
(*State IDLE*)
IF X_Act_St	= 0	THEN
	IF S_Trans_S0S10  THEN
		X_Act_St :=	10;
	END_IF
END_IF
(*State 10*)
IF X_Act_St = 10 THEN
  	IF S_Trans_S10S20 THEN		(*Transition from State 10 to State 20*)
  		X_Act_St := 20;
  	ELSIF S_Trans_S10S30 THEN	(*Transition from State 10 to State 30*)
  		X_Act_St := 30;
  	ELSIF S_Trans_S10S40 THEN	(*Transition from State 10 to State 40*)
  		X_Act_St := 40;
	ELSIF _FUN_Tools_TmOutStm(Tm_Actual:= Tm_Actual, Tm_Node_Entry:= Tm_Node_Entry, Tm_TmOut_Lmt:= T#10S)THEN 	(*Timeout state 10*)
		X_Act_St := 0;
	END_IF
(*State 20*)	
ELSIF X_Act_St = 20 THEN
  	IF S_Trans_S20S10 THEN		(*Transition from State 20 to State 10*)
  		X_Act_St := 10;
  	ELSIF S_Trans_S20S30 THEN		(*Transition from State 20 to State 30*)
  		X_Act_St := 30;
  	ELSIF S_Trans_S20S40 THEN		(*Transition from State 20 to State 40*)
  		X_Act_St := 40;
	ELSIF _FUN_Tools_TmOutStm(Tm_Actual:= Tm_Actual, Tm_Node_Entry:= Tm_Node_Entry, Tm_TmOut_Lmt:= T#10S)THEN	(*Timeout state 20*)
		X_Act_St := 0;
	END_IF
(*State 30*)
ELSIF X_Act_St = 30 THEN
  	IF S_Trans_S30S10 THEN		(*Transition from State 30 to State 10*)
  		X_Act_St := 10;
  	ELSIF S_Trans_S30S20 THEN		(*Transition from State 30 to State 20*)
  		X_Act_St := 20;
  	ELSIF S_Trans_S30S40 THEN		(*Transition from State 30 to State 40*)
  		X_Act_St := 40;
	ELSIF _FUN_Tools_TmOutStm(Tm_Actual:= Tm_Actual, Tm_Node_Entry:= Tm_Node_Entry, Tm_TmOut_Lmt:= T#10S)THEN	(*Timeout state 30*)
		X_Act_St := 0;
	END_IF
(*State 40*)
ELSIF X_Act_St = 40 THEN	
  	IF S_Trans_S40S10 THEN		(*Transition from State 40 to State 10*)
  		X_Act_St := 10;
  	ELSIF S_Trans_S40S20 THEN		(*Transition from State 40 to State 20*)
  		X_Act_St := 20;
  	ELSIF S_Trans_S40S30 THEN		(*Transition from State 40 to State 30*)
  		X_Act_St := 30;
	ELSIF _FUN_Tools_TmOutStm(Tm_Actual:= Tm_Actual, Tm_Node_Entry:= Tm_Node_Entry, Tm_TmOut_Lmt:= T#10S)THEN	(*Timeout state 40*)
		X_Act_St := 0;
	END_IF
END_IF
S_Idle	:=	(XActStat = 0);		(*Idle is active*)
S_Stat10 := (XActStat = 10);		(*State node is 10 active*)
S_Stat20 := (XActStat = 20);		(*State node is 20 active*)
S_Stat30 := (XActStat = 30);		(*State node is 30 active*)
S_Stat40 := (XActStat = 40);		(*State node is 40 active*)

S_New_Node := X_Act_Old <> X_Act_St;		(*Compare If the new node and old node is different*)


_FB_Tools_Shf_RegStm_01(C_Enable:= S_New_Node, X_Input:= X_Act_St);	(* save the state sequence in a shift register to debug the last 8 states *)
                  
END_FUNCTION_BLOCK

FUNCTION_BLOCK _FB_Tools_Comp_Hyst
  VAR_INPUT
    IN : REAL;
    UpTh : REAL;
    LoTh : REAL;
  END_VAR
  VAR_OUTPUT
    OUT : BOOL;
  END_VAR
  VAR
    POU_Version : WSTRING;
  END_VAR

                    (*
**********************************************************************
Bozankaya A.Ş.
**********************************************************************
Name					: _FB_Tools_Comp_Hyst
POU Type				: FB
Created by 				: E.TURKER , BZK.
Creation Date 			: 15-03-2022
Modifications			: see version description below


FB Description:
This FB handles compares the input data with a hysterysis.
For example
	An input value receives up on the high value, sets the outputs
	when the input value receives below the low value, reset the output.
*********************************************************************

Version 1	
*********************************************************************
Version Description:
- initial version
*********************************************************************
*)
POU_Version:="V0.1";
IF (IN > UpTh) THEN
	OUT := TRUE;
ELSIF (IN < LoTh) THEN
	OUT := FALSE;
END_IF;

                  
END_FUNCTION_BLOCK

FUNCTION_BLOCK _FB_Tools_ErrSet
  VAR_INPUT
    Trigger : BOOL := FALSE;
    Tm_Trig : TIME := TIME#0ms;
  END_VAR
  VAR_OUTPUT
    Event : BOOL := FALSE;
  END_VAR
  VAR
    FrcTrigger : BOOL := FALSE;
    TON_00 : TON;
    Disable : BOOL := FALSE;
    POU_version : WSTRING;
  END_VAR
  VAR  (* added by the conversion: wires and edge detectors of the diagram *)
    _OR5_OUT : BOOL;
  END_VAR

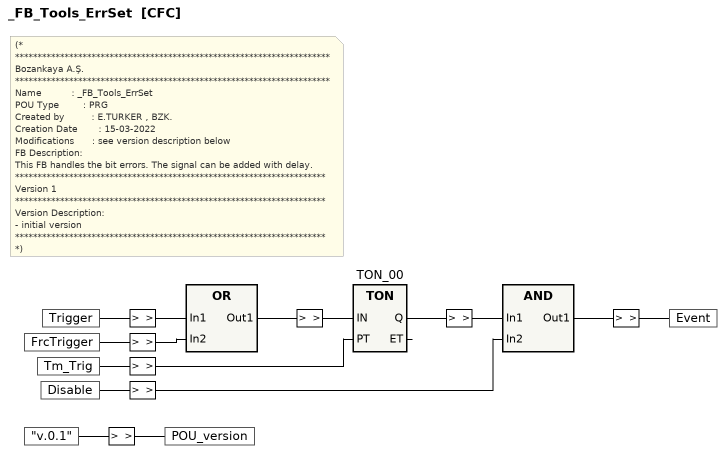
(* CFC diagram, written out as Structured Text *)
(* ( *
**********************************************************************
Bozankaya A.Ş.
**********************************************************************
Name					: _FB_Tools_ErrSet
POU Type				: PRG
Created by 				: E.TURKER , BZK.
Creation Date 			: 15-03-2022
Modifications			: see version description below


FB Description:
This FB handles the bit errors. The signal can be added with delay. 
*********************************************************************

Version 1	
*********************************************************************
Version Description:
- initial version
*********************************************************************
* ) *)
TON_00(IN := _OR5_OUT, PT := Tm_Trig);
POU_version := "v.0.1";
_OR5_OUT := Trigger OR FrcTrigger;
Event := TON_00.Q AND Disable;
END_FUNCTION_BLOCK

FUNCTION_BLOCK _FB_Tools_FrcHiLo
  VAR_INPUT
    S_Input : BOOL := FALSE;  (* Input signal *)
    C_FrcHi : BOOL := FALSE;
    C_FrcLo : BOOL := FALSE;
  END_VAR
  VAR_OUTPUT
    S_Output : BOOL := FALSE;  (* Output signal *)
  END_VAR
  VAR
    POU_version : WSTRING;
  END_VAR

                    (*
**********************************************************************
Bozankaya A.Ş.
**********************************************************************
Name					: _FB_Tools_FrcHiLo
POU Type				: FB
Created by 				: E.TURKER , BZK.
Creation Date 			: 15-03-2022
Modifications			: see version description below


FB Description:
This FB handles force high and low given input value.Basiclly force function
*********************************************************************

Version 1	
*********************************************************************
Version Description:
- initial version
*********************************************************************
*)
POU_Version:="V0.1";
IF NOT(C_FrcHi OR C_FrcLo) THEN		(*No Forcing variable*)
	S_Output	:=	S_Input;		
ELSIF C_FrcHi	THEN			(*Force TRUE If command is set*)
	S_Output	:=	TRUE;
ELSIF	C_FrcLo	THEN		(*Force FALSE If command is set*)
	S_Output	:=	FALSE;		
END_IF
                  
END_FUNCTION_BLOCK

FUNCTION_BLOCK _FB_Tools_Shf_RegStm
  VAR_INPUT
    C_Enable : BOOL;  (* Only active when new input set *)
    X_Input : UINT;  (* State machine active node *)
  END_VAR
  VAR_OUTPUT
    X_Old8 : UINT;  (* Oldest value *)
    X_Old7 : UINT;  (* ... *)
    X_Old6 : UINT;  (* ... *)
    X_Old5 : UINT;  (* ... *)
    X_Old4 : UINT;  (* ... *)
    X_Old3 : UINT;  (* ... *)
    X_Old2 : UINT;  (* ... *)
    X_Old1 : UINT;  (* Newest value *)
  END_VAR
  VAR
    POU_Version : WSTRING;
  END_VAR

                    (*
**********************************************************************
Bozankaya A.Ş.
**********************************************************************
Name					: _FB_Tools_Shf_RegStm
POU Type				: PRG
Created by 				: E.TURKER , BZK.
Creation Date 			: 16-03-2022
Modifications			: see version description below


FB Description:
This FB handles the store last 8 node state on state machines. Basiclly UINT Shift register
*********************************************************************

Version 1	
*********************************************************************
Version Description:
- initial version
*********************************************************************
*)
POU_Version:="V0.1";

IF C_Enable THEN
   X_Old8 := X_Old7;
   X_Old7 := X_Old6;
   X_Old6 := X_Old5;
   X_Old5 := X_Old4;
   X_Old4 := X_Old3;
   X_Old3 := X_Old2;
   X_Old2 := X_Old1;
   X_Old1 := X_Input;			(*assign new node and continue to shift when C_Enable given "TRUE" on the cycle*)
END_IF;
                  
END_FUNCTION_BLOCK

FUNCTION_BLOCK _FB_Tools_Toggle
  VAR_INPUT
    Input : BOOL;
    Reset : BOOL;
  END_VAR
  VAR_OUTPUT
    Output : BOOL;
  END_VAR
  VAR
    POU_version : WSTRING;
    P_C_FrcInput : BOOL;
    R_TRIG_00 : R_TRIG;
    RS_00 : RS;
    S_Output_Old : BOOL;
    P_C_Frc_Reset : BOOL;
  END_VAR
  VAR  (* added by the conversion: wires and edge detectors of the diagram *)
    _AND21_OUT : BOOL;
    _AND7_OUT : BOOL;
  END_VAR

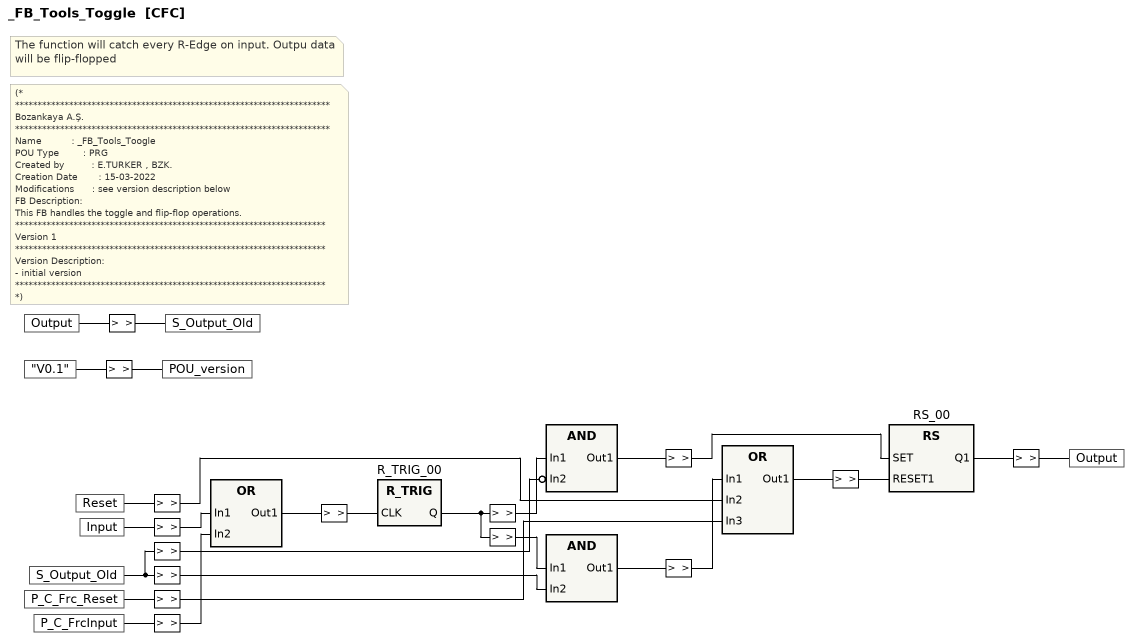
(* CFC diagram, written out as Structured Text *)
(* The function will catch every R-Edge on input. Outpu data will be flip-flopped *)
(* ( *
**********************************************************************
Bozankaya A.Ş.
**********************************************************************
Name					: _FB_Tools_Toogle
POU Type				: PRG
Created by 				: E.TURKER , BZK.
Creation Date 			: 15-03-2022
Modifications			: see version description below


FB Description:
This FB handles the toggle and flip-flop operations.
*********************************************************************

Version 1	
*********************************************************************
Version Description:
- initial version
*********************************************************************
* ) *)
Output := RS_00.Q1;
_AND21_OUT := R_TRIG_00.Q AND S_Output_Old;
RS_00(SET := _AND7_OUT, RESET1 := _AND21_OUT OR Reset OR P_C_Frc_Reset);
POU_version := "V0.1";
S_Output_Old := Output;
R_TRIG_00(CLK := Input OR P_C_FrcInput);
_AND7_OUT := R_TRIG_00.Q AND NOT S_Output_Old;
END_FUNCTION_BLOCK

FUNCTION_BLOCK _FB_UNPACK_BYTE_TO_8BITS
  VAR_INPUT
    X_BYTE_0 : BYTE;  (* Input WORD *)
  END_VAR
  VAR_OUTPUT
    S_BIT_0 : BOOL;  (* Less significant part *)
    S_BIT_1 : BOOL;
    S_BIT_2 : BOOL;
    S_BIT_3 : BOOL;
    S_BIT_4 : BOOL;
    S_BIT_5 : BOOL;
    S_BIT_6 : BOOL;
    S_BIT_7 : BOOL;  (* Most significant part *)
  END_VAR

                    S_BIT_0  := BYTE_TO_BOOL(X_BYTE_0 AND 2#00000001);					(*OR gate beginning from less significant part*)	
S_BIT_1  := BYTE_TO_BOOL(SHR(X_BYTE_0,1) AND 2#00000001);	
S_BIT_2  := BYTE_TO_BOOL(SHR(X_BYTE_0,2) AND 2#00000001);	
S_BIT_3  := BYTE_TO_BOOL(SHR(X_BYTE_0,3) AND 2#00000001);	
S_BIT_4  := BYTE_TO_BOOL(SHR(X_BYTE_0,4) AND 2#00000001);	
S_BIT_5  := BYTE_TO_BOOL(SHR(X_BYTE_0,5) AND 2#00000001);	
S_BIT_6  := BYTE_TO_BOOL(SHR(X_BYTE_0,6) AND 2#00000001);	
S_BIT_7  := BYTE_TO_BOOL(SHR(X_BYTE_0,7) AND 2#00000001);				(*OR gate ends with most significant part*)	
                  
END_FUNCTION_BLOCK

FUNCTION_BLOCK _FB_UNPACK_DWORD_TO_BYTE
  VAR_INPUT
    X_DWORD_0 : DWORD;  (* Input DWORD *)
  END_VAR
  VAR_OUTPUT
    X_BYTE_0 : BYTE;  (* Less significant part *)
    X_BYTE_1 : BYTE;
    X_BYTE_2 : BYTE;
    X_BYTE_3 : BYTE;  (* Most significant part *)
  END_VAR

                    X_BYTE_0:=DWORD_TO_BYTE(X_DWORD_0);					(*BYTE000000000000000000000000  <=   DWORD : *)
X_BYTE_1:=DWORD_TO_BYTE(SHR(X_DWORD_0,8));			(*00000000BYTE0000000000000000  <=   DWORD : *)
X_BYTE_2:=DWORD_TO_BYTE(SHR(X_DWORD_0,16));			(*0000000000000000BYTE00000000  <=   DWORD : *)
X_BYTE_3:=DWORD_TO_BYTE(SHR(X_DWORD_0,24));			(*000000000000000000000000BYTE  <=   DWORD : *)
                  
END_FUNCTION_BLOCK

FUNCTION_BLOCK _FB_UNPACK_DWORD_TO_WORD
  VAR_INPUT
    X_DWORD_0 : DWORD;  (* Input DWORD *)
  END_VAR
  VAR_OUTPUT
    X_WORD_0 : WORD;  (* Less significant part *)
    X_WORD_1 : WORD;  (* Most significant part *)
  END_VAR

                    X_WORD_0:=DWORD_TO_WORD(X_DWORD_0);					(*0000WORD  <=   DWORD : *)
X_WORD_1:=DWORD_TO_WORD(SHR(X_DWORD_0,16));			(*WORD0000  <=   DWORD : *)

                  
END_FUNCTION_BLOCK

FUNCTION_BLOCK _FB_UNPACK_LWORD_TO_BYTE
  VAR_INPUT
    X_LWORD_0 : LWORD;  (* Input DWORD *)
  END_VAR
  VAR_OUTPUT
    X_BYTE_0 : BYTE;  (* Less significant part *)
    X_BYTE_1 : BYTE;
    X_BYTE_2 : BYTE;
    X_BYTE_3 : BYTE;
    X_BYTE_4 : BYTE;
    X_BYTE_5 : BYTE;
    X_BYTE_6 : BYTE;
    X_BYTE_7 : BYTE;  (* Most significant part *)
  END_VAR

                    X_BYTE_0:=LWORD_TO_BYTE(X_LWORD_0);					
X_BYTE_1:=LWORD_TO_BYTE(SHR(X_LWORD_0,8));			
X_BYTE_2:=LWORD_TO_BYTE(SHR(X_LWORD_0,16));			
X_BYTE_3:=LWORD_TO_BYTE(SHR(X_LWORD_0,24));			
X_BYTE_4:=LWORD_TO_BYTE(SHR(X_LWORD_0,32));			
X_BYTE_5:=LWORD_TO_BYTE(SHR(X_LWORD_0,40));			
X_BYTE_6:=LWORD_TO_BYTE(SHR(X_LWORD_0,48));			
X_BYTE_7:=LWORD_TO_BYTE(SHR(X_LWORD_0,56));			
                  
END_FUNCTION_BLOCK

FUNCTION_BLOCK _FB_UNPACK_LWORD_TO_DWORD
  VAR_INPUT
    X_LWORD_0 : LWORD;  (* Input DWORD *)
  END_VAR
  VAR_OUTPUT
    X_DWORD_0 : DWORD;  (* Less significant part *)
    X_DWORD_1 : DWORD;  (* Most significant part *)
  END_VAR

                    X_DWORD_0:=LWORD_TO_DWORD(X_LWORD_0);					(*0000DWORD  <=   LWORD : *)
X_DWORD_1:=LWORD_TO_DWORD(SHR(X_LWORD_0,32));			(*DWORD0000  <=   LWORD : *)

                  
END_FUNCTION_BLOCK

FUNCTION_BLOCK _FB_UNPACK_WORD_TO_BYTE
  VAR_INPUT
    X_Word_0 : WORD;  (* Input WORD *)
  END_VAR
  VAR_OUTPUT
    X_Byte_0 : BYTE;  (* Less significant part *)
    X_Byte_1 : BYTE;  (* Most significant part *)
  END_VAR

                    X_Byte_0:=WORD_TO_BYTE(X_Word_0)		;					(*BYTE00000000  <=   WORD : *)
X_Byte_1:=WORD_TO_BYTE(SHR(X_Word_0,8))	;				(*00000000BYTE  <=   WORD : *)
                  
END_FUNCTION_BLOCK

FUNCTION _FUN_Tools_TmOutStm : BOOL
  VAR_INPUT
    Tm_Actual : TIME;
    Tm_Node_Entry : TIME;
    Tm_TmOut_Lmt : TIME := TIME#10s0ms;
  END_VAR
  VAR
    POU_Version : WSTRING;
  END_VAR

                    (*
**********************************************************************
Bozankaya A.Ş.
**********************************************************************
Name					: _FUN_Tools_TmOut
POU Type				: FUN
Created by 				: E.TURKER , BZK.
Creation Date 			: 16-03-2022
Modifications			: see version description below


FUN Description:
This FB handles the timeout operations. 
Tm_Actual -> Needs to be assigned every cycle.
Tm_Node_Entry -> Needs to be assign only node changed
Tm_TmOut_Lmt-> Time out parameter 
*********************************************************************

Version 1	
*********************************************************************
Version Description:
- initial version
*********************************************************************
*)

POU_Version	:="V0.1";

RETURN	((Tm_Actual - Tm_Node_Entry) > Tm_TmOut_Lmt);
                  
END_FUNCTION

PROGRAM P_IOVD_Param
  VAR
    _FB_CanTx_Message_Unpack_101 : _FB_CanTx_Message_Unpack;
    _FB_UNPACK_WORD_TO_BYTE_0 : _FB_UNPACK_WORD_TO_BYTE;
    _FB_UNPACK_BYTE_TO_8BITS_0 : _FB_UNPACK_BYTE_TO_8BITS;
    _FB_UNPACK_BYTE_TO_8BITS_1 : _FB_UNPACK_BYTE_TO_8BITS;
  END_VAR

                    //Added by Deniz Çıkış @17.10.2023
//-----------------------------------------------------------------------------------------------------------------------------

//MESSAGE------
{region " User Area : Parameter Send - ID:101"}

_FB_CanTx_Message_Unpack_101.X_Byte_0		:= USINT_TO_BYTE(REAL_TO_USINT((GVL.IOVD.X_Param_Arr.X_No)));
_FB_CanTx_Message_Unpack_101.X_Byte_1		:= USINT_TO_BYTE(REAL_TO_USINT((GVL.IOVD.X_Param_Arr.X_Usr_Id)));
	 
_FB_UNPACK_WORD_TO_BYTE_0( 	
							X_WORD_0:= UINT_TO_WORD(REAL_TO_UINT((GVL.IOVD.X_Param_Arr.X_Val))),
							X_BYTE_0=> _FB_CanTx_Message_Unpack_101.X_Byte_2,
							X_BYTE_1=> _FB_CanTx_Message_Unpack_101.X_Byte_3);
								 
_FB_CanTx_Message_Unpack_101.X_Byte_4		:= USINT_TO_BYTE(REAL_TO_USINT((GVL.IOVD.X_Param_Arr.X_Days)));
	 
_FB_UNPACK_BYTE_TO_8BITS_0(
							S_Bit_0=> _FB_CanTx_Message_Unpack_101.S_Bit_40,
							S_Bit_1=> _FB_CanTx_Message_Unpack_101.S_Bit_41 ,
							S_Bit_2=> _FB_CanTx_Message_Unpack_101.S_Bit_42 ,
							S_Bit_3=> _FB_CanTx_Message_Unpack_101.S_Bit_43 ,
							X_BYTE_0:= USINT_TO_BYTE(REAL_TO_USINT((GVL.IOVD.X_Param_Arr.X_Months))));
								 
_FB_UNPACK_BYTE_TO_8BITS_1(
							S_Bit_0=> _FB_CanTx_Message_Unpack_101.S_Bit_44,
							S_Bit_1=> _FB_CanTx_Message_Unpack_101.S_Bit_45 ,
							S_Bit_2=> _FB_CanTx_Message_Unpack_101.S_Bit_46 ,
							S_Bit_3=> _FB_CanTx_Message_Unpack_101.S_Bit_47 ,
							X_BYTE_0:= USINT_TO_BYTE(REAL_TO_USINT((GVL.IOVD.X_Param_Arr.X_Years))));		

_FB_CanTx_Message_Unpack_101.X_Byte_6		:= USINT_TO_BYTE(REAL_TO_USINT((GVL.IOVD.X_Param_Arr.X_Hours)));	
_FB_CanTx_Message_Unpack_101.X_Byte_7		:= USINT_TO_BYTE(REAL_TO_USINT((GVL.IOVD.X_Param_Arr.X_Minutes)));	

_FB_CanTx_Message_Unpack_101(
     C_Enable:= NOT GVL.IIVD.S_TmOut_Diag_Temel_Durum_0X300 AND GVL.IIVD.S_Para_Pg_Act.x AND GVL.IIVD.C_Par_Rx.x AND NOT GVL.IIVD.C_Par_Wr.x,
     Obj_CAN:= ADR(GVL.IC.Obj_CAN0),
     X_MsgID:= 16#101,
     Tm_CycleTime:= TIME#50MS,
     N_Msg_Dlc:=8,
     S_Extended:= 0,
     S_Sent_Ok   => GVL.IOVD.S_SentOk_Parametre_0X101);					  
                  
END_PROGRAM

(* PR1006_REV_002449_TIMTRO, Serdar Temeltaşı @19.06.2025 Araçta pantograf şarjı aktif durumunun oluşturulması için TCU'dan alınarak kullanılan; 0x18FFE2EF grubundaki "pantograf şarj durumu" ve "pantograf şarj kontaktörü durumu" sinyalleri yerine, "pantograf yukarıda" ve "batarya konvertörü aktif" durumları kontrol edildi. PR1006_REV_002726_TIMTRO, Serdar Temeltaşı @17.07.2025 DWP'ye gönderilen kırmızı batarya hatası MBMS'den alınan "kırmızı lamba" sinyalinin aktif olması durumunda DWP'ye gönderilen kırmızı batarya hatası, "sarı lamba" sinyalinin aktif olması durumunda ise DWP'ye gönderilen sarı batarya hatasının aktif edilmesi sağlandı. PR1006_REV_002727_TIMTRO, Serdar Temeltaşı @17.07.2025 DWP'ye batarya akımı değerinin gönderilebilmesi için yüksek voltaj aktivasyon işlemlerinin başlatılıp başlatılmadığı kontrol edildi. *)
PROGRAM P_IOVD_B
  VAR
    _FB_CanTx_Message_Unpack_430 : _FB_CanTx_Message_Unpack;
    _FB_CanTx_Message_Unpack_431 : _FB_CanTx_Message_Unpack;
    _FB_CanTx_Message_432 : _FB_CanTx_Message;
    _FB_CanTx_Message_433 : _FB_CanTx_Message;
    _FB_CanTx_Message_Unpack_434 : _FB_CanTx_Message_Unpack;
    _FB_CanTx_Message_435 : _FB_CanTx_Message;
    _FB_CanTx_Message_436 : _FB_CanTx_Message;
    _FB_CanTx_Message_Unpack_437 : _FB_CanTx_Message_Unpack;
    _FB_CanTx_Message_438 : _FB_CanTx_Message;
    _FB_CanTx_Message_Unpack_4A0 : _FB_CanTx_Message_Unpack;
    _FB_CanTx_Message_Unpack_4A5 : _FB_CanTx_Message_Unpack;
    _FB_CanTx_Message_Unpack_4A6 : _FB_CanTx_Message_Unpack;
    _FB_CanTx_Message_Unpack_4AF : _FB_CanTx_Message_Unpack;
    _FB_CanTx_Message_Unpack_4F0 : _FB_CanTx_Message_Unpack;
    _FB_UNPACK_WORD_TO_BYTE_0 : _FB_UNPACK_WORD_TO_BYTE;
    _FB_UNPACK_WORD_TO_BYTE_1 : _FB_UNPACK_WORD_TO_BYTE;
    _FB_UNPACK_WORD_TO_BYTE_2 : _FB_UNPACK_WORD_TO_BYTE;
    _FB_UNPACK_WORD_TO_BYTE_3 : _FB_UNPACK_WORD_TO_BYTE;
    _FB_UNPACK_WORD_TO_BYTE_4 : _FB_UNPACK_WORD_TO_BYTE;
    _FB_UNPACK_WORD_TO_BYTE_5 : _FB_UNPACK_WORD_TO_BYTE;
    _FB_UNPACK_WORD_TO_BYTE_6 : _FB_UNPACK_WORD_TO_BYTE;
    _FB_UNPACK_WORD_TO_BYTE_7 : _FB_UNPACK_WORD_TO_BYTE;
    _FB_UNPACK_WORD_TO_BYTE_8 : _FB_UNPACK_WORD_TO_BYTE;
    _FB_UNPACK_WORD_TO_BYTE_9 : _FB_UNPACK_WORD_TO_BYTE;
    _FB_UNPACK_WORD_TO_BYTE_10 : _FB_UNPACK_WORD_TO_BYTE;
    _FB_UNPACK_WORD_TO_BYTE_11 : _FB_UNPACK_WORD_TO_BYTE;
    _FB_UNPACK_WORD_TO_BYTE_12 : _FB_UNPACK_WORD_TO_BYTE;
    _FB_UNPACK_WORD_TO_BYTE_13 : _FB_UNPACK_WORD_TO_BYTE;
    _FB_UNPACK_WORD_TO_BYTE_14 : _FB_UNPACK_WORD_TO_BYTE;
    _FB_UNPACK_WORD_TO_BYTE_15 : _FB_UNPACK_WORD_TO_BYTE;
    _FB_UNPACK_WORD_TO_BYTE_16 : _FB_UNPACK_WORD_TO_BYTE;
    _FB_UNPACK_WORD_TO_BYTE_17 : _FB_UNPACK_WORD_TO_BYTE;
    _FB_UNPACK_WORD_TO_BYTE_18 : _FB_UNPACK_WORD_TO_BYTE;
    _FB_UNPACK_WORD_TO_BYTE_19 : _FB_UNPACK_WORD_TO_BYTE;
    _FB_UNPACK_WORD_TO_BYTE_20 : _FB_UNPACK_WORD_TO_BYTE;
    _FB_UNPACK_WORD_TO_BYTE_21 : _FB_UNPACK_WORD_TO_BYTE;
    _FB_UNPACK_WORD_TO_BYTE_22 : _FB_UNPACK_WORD_TO_BYTE;
    _FB_UNPACK_WORD_TO_BYTE_23 : _FB_UNPACK_WORD_TO_BYTE;
    _FB_UNPACK_WORD_TO_BYTE_24 : _FB_UNPACK_WORD_TO_BYTE;
    _FB_UNPACK_WORD_TO_BYTE_25 : _FB_UNPACK_WORD_TO_BYTE;
    _FB_UNPACK_BYTE_TO_8BITS_0 : _FB_UNPACK_BYTE_TO_8BITS;
    _FB_UNPACK_BYTE_TO_8BITS_10 : _FB_UNPACK_BYTE_TO_8BITS;
    _FB_UNPACK_BYTE_TO_8BITS_23 : _FB_UNPACK_BYTE_TO_8BITS;
    _FB_PACK_8BITS_TO_BYTE_0 : _FB_PACK_8BITS_TO_BYTE;
    _FB_PACK_8BITS_TO_BYTE_1 : _FB_PACK_8BITS_TO_BYTE;
    _FB_PACK_8BITS_TO_BYTE_2 : _FB_PACK_8BITS_TO_BYTE;
  END_VAR

                    (*
**********************************************************************
Bozankaya A.Ş.
**********************************************************************
Name					: P_IOVD_B
POU Type				: Program
Created by              : COMMUNICATION INTERFACE GENERATOR V1.1.034(denizcikispc), BZK.
Creation Date 			: 2023-07-11T10:33:11
Modifications			: see version description below


Program Description:This program which is created by automatically by communication interface generator 
 handles the TX (OUTPUT) can messages according to CAN_500_LIB 
*********************************************************************

Version 1	
*********************************************************************
Version Description:
- initial version
*********************************************************************
*)
//-----------------------------------------------------------------------------------------------------------------------------
//MESSAGE------
{region " User Area : ESS_Durum- ID:430"}

//-------SIGNAL -> S_ESS_Mn_Ct Max: 1 Min: 0 Def: 0 Resolution: 1 Offset: 0
GVL.IOVD.S_ESS_Mn_Ct.v					:= GVL.SY.S_ECU_Rdy AND NOT GVL.IOVD.S_ESS_Mn_Ct.e AND NOT GVL.IOVD.S_ESS_Mn_Ct.na;
GVL.IOVD.S_ESS_Mn_Ct.x					:= GVL.IIME.S_Mn_Ct.x;
GVL.IOVD.S_ESS_Mn_Ct.e					:= GVL.IIME.S_Mn_Ct.e;
GVL.IOVD.S_ESS_Mn_Ct.na					:= GVL.IIME.S_Mn_Ct.na;
//-------SIGNAL -> S_Insu_Ok Max: 1 Min: 0 Def: 0 Resolution: 1 Offset: 0
GVL.IOVD.S_Insu_Ok.v					:= GVL.SY.S_ECU_Rdy AND NOT GVL.IOVD.S_Insu_Ok.e AND NOT GVL.IOVD.S_Insu_Ok.na;
GVL.IOVD.S_Insu_Ok.x					:= GVL.IIME.S_Int_Insu.x;
GVL.IOVD.S_Insu_Ok.e					:= GVL.IIME.S_Int_Insu.e;
GVL.IOVD.S_Insu_Ok.na					:= GVL.IIME.S_Int_Insu.na;
//-------SIGNAL -> S_BMS_Sp Max: 1 Min: 0 Def: 0 Resolution: 1 Offset: 0
GVL.IOVD.S_BMS_Sp.v						:= GVL.SY.S_ECU_Rdy AND NOT GVL.IOVD.S_BMS_Sp.e AND NOT GVL.IOVD.S_BMS_Sp.na;
GVL.IOVD.S_BMS_Sp.x						:= NOT GVL.IIME.S_Com_Flt;
GVL.IOVD.S_BMS_Sp.e						:= FALSE;
GVL.IOVD.S_BMS_Sp.na					:= FALSE;
//-------SIGNAL -> S_Bat_Mode Max: 1 Min: 0 Def: 0 Resolution: 1 Offset: 0
GVL.IOVD.S_Bat_Mode.v					:= GVL.SY.S_ECU_Rdy AND NOT GVL.IOVD.S_Bat_Mode.e AND NOT GVL.IOVD.S_Bat_Mode.na;
GVL.IOVD.S_Bat_Mode.x					:= GVL.IIPT.S_Bat_Mod_Stat.x;
GVL.IOVD.S_Bat_Mode.e					:= GVL.IIPT.S_Bat_Mod_Stat.e;
GVL.IOVD.S_Bat_Mode.na					:= GVL.IIPT.S_Bat_Mod_Stat.na;
//-------SIGNAL -> S_Ops_Mode Max: 1 Min: 0 Def: 0 Resolution: 1 Offset: 0
GVL.IOVD.S_Ops_Mode.v					:= GVL.SY.S_ECU_Rdy AND NOT GVL.IOVD.S_Ops_Mode.e AND NOT GVL.IOVD.S_Ops_Mode.na;
GVL.IOVD.S_Ops_Mode.x					:= GVL.IIME.Z_Bat_Sys_Ops_Mode.x = 2;
GVL.IOVD.S_Ops_Mode.e					:= GVL.IIME.S_Com_Distrb;
GVL.IOVD.S_Ops_Mode.na					:= FALSE;
//-------SIGNAL -> C_Tr_Mode Max: 1 Min: 0 Def: 0 Resolution: 1 Offset: 0
GVL.IOVD.C_Tr_Mode.v					:= GVL.SY.S_ECU_Rdy AND NOT GVL.IOVD.C_Tr_Mode.e AND NOT GVL.IOVD.C_Tr_Mode.na;
GVL.IOVD.C_Tr_Mode.x					:= GVL.IOME.Z_Vh_Mode_Req.x = 3;
GVL.IOVD.C_Tr_Mode.e					:= GVL.IOME.Z_Vh_Mode_Req.e;
GVL.IOVD.C_Tr_Mode.na					:= GVL.IOME.Z_Vh_Mode_Req.na;
//-------SIGNAL -> S_Pwr_Distr Max: 1 Min: 0 Def: 0 Resolution: 1 Offset: 0
GVL.IOVD.S_Pwr_Distr.v					:= GVL.SY.S_ECU_Rdy AND NOT GVL.IOVD.S_Pwr_Distr.e AND NOT GVL.IOVD.S_Pwr_Distr.na;
GVL.IOVD.S_Pwr_Distr.x					:= GVL.ME.S_ESS_Ops_Mode AND GVL.IIME.X_I_Act_Bat.x <> 0;
GVL.IOVD.S_Pwr_Distr.e					:= GVL.IIME.S_Com_Flt OR GVL.IIME.X_I_Act_Bat.e;
GVL.IOVD.S_Pwr_Distr.na					:= GVL.IIME.X_I_Act_Bat.na;
//-------SIGNAL -> S_Ext_Sp_Req Max: 1 Min: 0 Def: 0 Resolution: 1 Offset: 0
GVL.IOVD.S_Ext_Sp_Req.v					:= GVL.SY.S_ECU_Rdy AND NOT GVL.IOVD.S_Ext_Sp_Req.e AND NOT GVL.IOVD.S_Ext_Sp_Req.na;
GVL.IOVD.S_Ext_Sp_Req.x					:= GVL.IOME.Z_Ext_Engy_Conn_Req.x = 1;
GVL.IOVD.S_Ext_Sp_Req.e					:= GVL.IOME.Z_Ext_Engy_Conn_Req.e;
GVL.IOVD.S_Ext_Sp_Req.na				:= GVL.IOME.Z_Ext_Engy_Conn_Req.na;
//-------SIGNAL -> S_Vh_Mode_Req Max: 1 Min: 0 Def: 0 Resolution: 1 Offset: 0
GVL.IOVD.X_Vh_Mode_Req.v				:= GVL.SY.S_ECU_Rdy AND NOT GVL.IOVD.X_Vh_Mode_Req.e AND NOT GVL.IOVD.X_Vh_Mode_Req.na;
GVL.IOVD.X_Vh_Mode_Req.x				:= GVL.IOME.Z_Vh_Mode_Req.x;
GVL.IOVD.X_Vh_Mode_Req.e				:= GVL.IOME.Z_Vh_Mode_Req.e;
GVL.IOVD.X_Vh_Mode_Req.na				:= GVL.IOME.Z_Vh_Mode_Req.na;
//-------SIGNAL -> Z_MBMS_Mode Max: 250 Min: 0 Def: 0 Resolution: 1 Offset: 0
GVL.IOVD.Z_MBMS_Mode.v					:= GVL.SY.S_ECU_Rdy AND NOT GVL.IOVD.Z_MBMS_Mode.e AND NOT GVL.IOVD.Z_MBMS_Mode.na;
GVL.IOVD.Z_MBMS_Mode.x					:= GVL.IIME.Z_Bat_Sys_Avl_Mode.x;
GVL.IOVD.Z_MBMS_Mode.e					:= GVL.IIME.Z_Bat_Sys_Avl_Mode.e;
GVL.IOVD.Z_MBMS_Mode.na					:= GVL.IIME.Z_Bat_Sys_Avl_Mode.na;
GVL.IOVD.Z_MBMS_Mode.RangeExcd			:= (250 < GVL.IOVD.Z_MBMS_Mode.x) OR (0 > GVL.IOVD.Z_MBMS_Mode.x);
//-------SIGNAL -> Z_Bat_Ops Max: 15 Min: 0 Def: 0 Resolution: 1 Offset: 0
GVL.IOVD.Z_Bat_Ops.v					:= GVL.SY.S_ECU_Rdy AND NOT GVL.IOVD.Z_Bat_Ops.e AND NOT GVL.IOVD.Z_Bat_Ops.na;
GVL.IOVD.Z_Bat_Ops.x					:= GVL.IIME.Z_Bat_Sys_Ops_Mode.x;
GVL.IOVD.Z_Bat_Ops.e					:= GVL.IIME.Z_Bat_Sys_Ops_Mode.e;
GVL.IOVD.Z_Bat_Ops.na					:= GVL.IIME.Z_Bat_Sys_Ops_Mode.na;
GVL.IOVD.Z_Bat_Ops.RangeExcd			:= (15 < GVL.IOVD.Z_Bat_Ops.x) OR (0 > GVL.IOVD.Z_Bat_Ops.x);
//-------SIGNAL -> C_BMS_Wkup Max: 1 Min: 0 Def: 0 Resolution: 1 Offset: 0
GVL.IOVD.C_BMS_Wkup.v					:= TRUE;
GVL.IOVD.C_BMS_Wkup.x					:= GVL.IORE.C_MBMS_Wkup;
//-------SIGNAL -> Z_Bat_Mode Max: 250 Min: 0 Def: 0 Resolution: 1 Offset: 0
GVL.IOVD.Z_Bat_Mode.v					:= GVL.SY.S_ECU_Rdy AND NOT GVL.IOVD.Z_Bat_Mode.e AND NOT GVL.IOVD.Z_Bat_Mode.na;
GVL.IOVD.Z_Bat_Mode.x					:= GVL.IIME.Z_Bat_Sys_Ops_Mode.x;
GVL.IOVD.Z_Bat_Mode.e					:= GVL.IIME.Z_Bat_Sys_Ops_Mode.e;
GVL.IOVD.Z_Bat_Mode.na					:= GVL.IIME.Z_Bat_Sys_Ops_Mode.na;
GVL.IOVD.Z_Bat_Mode.RangeExcd			:=  (250 < GVL.IOVD.Z_Bat_Mode.x) OR (0 > GVL.IOVD.Z_Bat_Mode.x);
//-------SIGNAL -> Z_ESS_Stat Max: 255 Min: 0 Def: 0 Resolution: 1 Offset: 0
GVL.IOVD.Z_ESS_Stat.v					:= GVL.SY.S_ECU_Rdy AND NOT GVL.IOVD.Z_ESS_Stat.e AND NOT GVL.IOVD.Z_ESS_Stat.na;
_FB_PACK_8BITS_TO_BYTE_1 (	S_BIT_0 	:= GVL.IIME.Z_Bat_Sys_Ops_Mode.x = 2 AND GVL.IIME.X_Pac_Onl.x > 0,
							S_BIT_1		:= BYTE_TO_BOOL(GVL.IIME.S_MBMS_Lmp_Red.x),				// PR1006_REV_002726_TIMTRO
							S_BIT_2 	:= BYTE_TO_BOOL(GVL.IIME.S_MBMS_Lmp_Amb.x),				// PR1006_REV_002726_TIMTRO
							S_BIT_3 	:= (GVL.IIMP.Z_Pnt_Stat.x = 2 AND GVL.IIPT.S_Bat_Cnv_Stat.x AND GVL.IIME.X_I_Act_Bat.x < 0),
							S_BIT_4 	:= GVL.IIPT.S_Bat_Mod_Stat.x AND GVL.IIME.Z_Bat_Sys_Ops_Mode.x = 1,
							S_BIT_5 	:= GVL.PV.S_Lo_SOC_Amb,
							S_BIT_6 	:= GVL.PV.S_Lo_SOC_Red,
							S_BIT_7 	:= 0,
							X_BYTE_0 	=> GVL.IOVD.Z_ESS_Stat.x);
GVL.IOVD.Z_ESS_Stat.e					:= FALSE;
GVL.IOVD.Z_ESS_Stat.na					:= FALSE;
GVL.IOVD.Z_ESS_Stat.RangeExcd			:= (255 < GVL.IOVD.Z_ESS_Stat.x) OR (0 > GVL.IOVD.Z_ESS_Stat.x);
{endregion}
//-----------------------------------------------------------------------------------------------------------------------------
//-----------------------------------------------------------------------------------------------------------------------------
//MESSAGE------
{region " User Area : ESS_Paket_Voltaji- ID:431"}
//-------SIGNAL -> X_U_Bat_1 Max: 1300 Min: 0 Def: 0 Resolution: 0.02 Offset: 0
GVL.IOVD.X_U_Bat_1.v					:= GVL.SY.S_ECU_Rdy AND NOT GVL.IOVD.X_U_Bat_1.e AND NOT GVL.IOVD.X_U_Bat_1.na AND NOT GVL.IOVD.X_U_Bat_1.RangeExcd;
GVL.IOVD.X_U_Bat_1.x					:= GVL.IIME.X_U_Act_Bat.x; 
GVL.IOVD.X_U_Bat_1.e					:= GVL.IIME.X_U_Act_Bat.e;
GVL.IOVD.X_U_Bat_1.na					:= GVL.IIME.X_U_Act_Bat.na;
GVL.IOVD.X_U_Bat_1.RangeExcd			:= (1300 < GVL.IOVD.X_U_Bat_1.x) OR (0 > GVL.IOVD.X_U_Bat_1.x);
//-------SIGNAL -> X_U_Bat_2 Max: 1300 Min: 0 Def: 0 Resolution: 0.02 Offset: 0
GVL.IOVD.X_U_Bat_2.v					:= GVL.SY.S_ECU_Rdy AND NOT GVL.IOVD.X_U_Bat_2.e AND NOT GVL.IOVD.X_U_Bat_2.na AND NOT GVL.IOVD.X_U_Bat_2.RangeExcd;
GVL.IOVD.X_U_Bat_2.x					:= GVL.IIME.X_U_Act_Bat.x; 
GVL.IOVD.X_U_Bat_2.e					:= GVL.IIME.X_U_Act_Bat.e; 
GVL.IOVD.X_U_Bat_2.na					:= GVL.IIME.X_U_Act_Bat.na;
GVL.IOVD.X_U_Bat_2.RangeExcd			:= (1300 < GVL.IOVD.X_U_Bat_2.x) OR (0 > GVL.IOVD.X_U_Bat_2.x);
//-------SIGNAL -> X_U_Bat_3 Max: 1300 Min: 0 Def: 0 Resolution: 0.02 Offset: 0
// GVL.IOVD.X_U_Bat_3.v					:= GVL.SY.S_ECU_Rdy AND NOT GVL.IOVD.X_U_Bat_3.e AND NOT GVL.IOVD.X_U_Bat_3.na AND NOT GVL.IOVD.X_U_Bat_3.RangeExcd;
// GVL.IOVD.X_U_Bat_3.x					:= GVL.IIMEP.X_U_Cell_Pac_3.x; 
// GVL.IOVD.X_U_Bat_3.e					:= GVL.IIMEP.X_U_Cell_Pac_3.e; 
// GVL.IOVD.X_U_Bat_3.na					:= GVL.IIMEP.X_U_Cell_Pac_3.na;
// GVL.IOVD.X_U_Bat_3.RangeExcd			:= (1300 < GVL.IOVD.X_U_Bat_3.x) OR (0 > GVL.IOVD.X_U_Bat_3.x);
//-------SIGNAL -> X_U_Bat_4 Max: 1300 Min: 0 Def: 0 Resolution: 0.02 Offset: 0
GVL.IOVD.X_U_Bat_4.v					:= GVL.SY.S_ECU_Rdy AND NOT GVL.IOVD.X_U_Bat_4.e AND NOT GVL.IOVD.X_U_Bat_4.na AND NOT GVL.IOVD.X_U_Bat_4.RangeExcd;
GVL.IOVD.X_U_Bat_4.x					:= 0;
GVL.IOVD.X_U_Bat_4.e					:= FALSE;
GVL.IOVD.X_U_Bat_4.na					:= FALSE;
GVL.IOVD.X_U_Bat_4.RangeExcd			:= (1300 < GVL.IOVD.X_U_Bat_4.x) OR (0 > GVL.IOVD.X_U_Bat_4.x);
{endregion}
//-----------------------------------------------------------------------------------------------------------------------------
//-----------------------------------------------------------------------------------------------------------------------------
//MESSAGE------
{region " User Area : ESS_Paket_Akim- ID:432"}

//-------SIGNAL -> X_I_Bat_1 Max: 3000 Min: -3000 Def: 0 Resolution: 0.1 Offset: -3276.8
GVL.IOVD.X_I_Bat_1.v					:= GVL.SY.S_ECU_Rdy AND GVL.ME.S_HV_En AND NOT GVL.IOVD.X_I_Bat_1.e AND NOT GVL.IOVD.X_I_Bat_1.na AND NOT GVL.IOVD.X_I_Bat_1.RangeExcd;		// PR1006_REV_002727_TIMTRO
GVL.IOVD.X_I_Bat_1.x					:= GVL.IIME.X_I_Act_Bat.x;
GVL.IOVD.X_I_Bat_1.e					:= GVL.IIME.X_I_Act_Bat.e;
GVL.IOVD.X_I_Bat_1.na					:= GVL.IIME.X_I_Act_Bat.na;
GVL.IOVD.X_I_Bat_1.RangeExcd			:= (3000 < GVL.IOVD.X_I_Bat_1.x) OR (-3000 > GVL.IOVD.X_I_Bat_1.x);
//-------SIGNAL -> X_I_Bat_2 Max: 3000 Min: -3000 Def: 0 Resolution: 0.1 Offset: -3276.8
GVL.IOVD.X_I_Bat_2.v					:= GVL.SY.S_ECU_Rdy AND GVL.ME.S_HV_En AND NOT GVL.IOVD.X_I_Bat_2.e AND NOT GVL.IOVD.X_I_Bat_2.na AND NOT GVL.IOVD.X_I_Bat_2.RangeExcd;
GVL.IOVD.X_I_Bat_2.x					:= GVL.IIME.X_I_Act_Bat.x;
GVL.IOVD.X_I_Bat_2.e					:= GVL.IIME.X_I_Act_Bat.e;
GVL.IOVD.X_I_Bat_2.na					:= GVL.IIME.X_I_Act_Bat.na;
GVL.IOVD.X_I_Bat_2.RangeExcd			:= (3000 < GVL.IOVD.X_I_Bat_2.x) OR (-3000 > GVL.IOVD.X_I_Bat_2.x);
//-------SIGNAL -> X_I_Bat_3 Max: 3000 Min: -3000 Def: 0 Resolution: 0.1 Offset: -3276.8
GVL.IOVD.X_I_Bat_3.v					:= GVL.SY.S_ECU_Rdy AND GVL.ME.S_HV_En AND NOT GVL.IOVD.X_I_Bat_3.e AND NOT GVL.IOVD.X_I_Bat_3.na AND NOT GVL.IOVD.X_I_Bat_3.RangeExcd;
GVL.IOVD.X_I_Bat_3.x					:= GVL.IIME.X_I_Act_Bat.x;
GVL.IOVD.X_I_Bat_3.e					:= GVL.IIME.X_I_Act_Bat.e;
GVL.IOVD.X_I_Bat_3.na					:= GVL.IIME.X_I_Act_Bat.na;
GVL.IOVD.X_I_Bat_3.RangeExcd			:= (3000 < GVL.IOVD.X_I_Bat_3.x) OR (-3000 > GVL.IOVD.X_I_Bat_3.x);
//-------SIGNAL -> X_I_Bat_4 Max: 3000 Min: -3000 Def: 0 Resolution: 0.1 Offset: -3276.8
GVL.IOVD.X_I_Bat_4.v					:= GVL.SY.S_ECU_Rdy AND GVL.ME.S_HV_En AND NOT GVL.IOVD.X_I_Bat_4.e AND NOT GVL.IOVD.X_I_Bat_4.na AND NOT GVL.IOVD.X_I_Bat_4.RangeExcd;
GVL.IOVD.X_I_Bat_4.x					:= 0;
GVL.IOVD.X_I_Bat_4.e					:= FALSE;
GVL.IOVD.X_I_Bat_4.na					:= FALSE;
GVL.IOVD.X_I_Bat_4.RangeExcd			:= (3000 < GVL.IOVD.X_I_Bat_4.x) OR (-3000 > GVL.IOVD.X_I_Bat_4.x);
{endregion}
//-----------------------------------------------------------------------------------------------------------------------------
//-----------------------------------------------------------------------------------------------------------------------------
//MESSAGE------
{region " User Area : ESS_Maksimum_Hucre_Voltaji- ID:433"}

//-------SIGNAL -> X_U_Max_Cell_1 Max: 4 Min: 0 Def: 0 Resolution: 0.01 Offset: 0
GVL.IOVD.X_U_Max_Bat_1.v					:= GVL.SY.S_ECU_Rdy AND NOT GVL.IOVD.X_U_Max_Bat_1.e AND NOT GVL.IOVD.X_U_Max_Bat_1.na;
GVL.IOVD.X_U_Max_Bat_1.x					:= GVL.IIME.X_U_Max_Act_Bat.x;
GVL.IOVD.X_U_Max_Bat_1.e					:= GVL.IIME.X_U_Max_Act_Bat.e;
GVL.IOVD.X_U_Max_Bat_1.na					:= GVL.IIME.X_U_Max_Act_Bat.na;
GVL.IOVD.X_U_Max_Bat_1.RangeExcd			:= (850 < GVL.IOVD.X_U_Max_Bat_1.x) OR (0 > GVL.IOVD.X_U_Max_Bat_1.x);
//-------SIGNAL -> X_U_Max_Cell_2 Max: 4 Min: 0 Def: 0 Resolution: 0.01 Offset: 0
GVL.IOVD.X_U_Max_Bat_2.v					:= GVL.SY.S_ECU_Rdy AND NOT GVL.IOVD.X_U_Max_Bat_2.e AND NOT GVL.IOVD.X_U_Max_Bat_2.na;
GVL.IOVD.X_U_Max_Bat_2.x					:= GVL.IIME.X_U_Max_Act_Bat.x;
GVL.IOVD.X_U_Max_Bat_2.e					:= GVL.IIME.X_U_Max_Act_Bat.e;
GVL.IOVD.X_U_Max_Bat_2.na					:= GVL.IIME.X_U_Max_Act_Bat.na;
GVL.IOVD.X_U_Max_Bat_2.RangeExcd			:= (850 < GVL.IOVD.X_U_Max_Bat_2.x) OR (0 > GVL.IOVD.X_U_Max_Bat_2.x);
//-------SIGNAL -> X_U_Max_Cell_3 Max: 4 Min: 0 Def: 0 Resolution: 0.01 Offset: 0
GVL.IOVD.X_U_Max_Bat_3.v					:= GVL.SY.S_ECU_Rdy AND NOT GVL.IOVD.X_U_Max_Bat_3.e AND NOT GVL.IOVD.X_U_Max_Bat_3.na;
GVL.IOVD.X_U_Max_Bat_3.x					:= GVL.IIME.X_U_Max_Act_Bat.x;
GVL.IOVD.X_U_Max_Bat_3.e					:= GVL.IIME.X_U_Max_Act_Bat.e;
GVL.IOVD.X_U_Max_Bat_3.na					:= GVL.IIME.X_U_Max_Act_Bat.na;
GVL.IOVD.X_U_Max_Bat_3.RangeExcd			:= (850 < GVL.IOVD.X_U_Max_Bat_3.x) OR (0 > GVL.IOVD.X_U_Max_Bat_3.x);
//-------SIGNAL -> X_U_Max_Cell_4 Max: 4 Min: 0 Def: 0 Resolution: 0.01 Offset: 0
GVL.IOVD.X_U_Max_Bat_4.v					:= GVL.SY.S_ECU_Rdy AND NOT GVL.IOVD.X_U_Max_Bat_4.e AND NOT GVL.IOVD.X_U_Max_Bat_4.na;
GVL.IOVD.X_U_Max_Bat_4.x					:= GVL.IIME.X_U_Max_Act_Bat.x;
GVL.IOVD.X_U_Max_Bat_4.e					:= GVL.IIME.X_U_Max_Act_Bat.e;
GVL.IOVD.X_U_Max_Bat_4.na					:= GVL.IIME.X_U_Max_Act_Bat.na;
GVL.IOVD.X_U_Max_Bat_4.RangeExcd			:= (850 < GVL.IOVD.X_U_Max_Bat_4.x) OR (0 > GVL.IOVD.X_U_Max_Bat_4.x);
{endregion}
//-----------------------------------------------------------------------------------------------------------------------------
//-----------------------------------------------------------------------------------------------------------------------------
//MESSAGE------
{region " User Area : ESS_Minimum_Hucre_Voltaji- ID:434"}

//-------SIGNAL -> X_U_Min_Cell_1 Max: 4 Min: 0 Def: 0 Resolution: 0.01 Offset: 0
GVL.IOVD.X_U_Min_Bat_1.v					:= GVL.SY.S_ECU_Rdy AND NOT GVL.IOVD.X_U_Min_Bat_1.e AND NOT GVL.IOVD.X_U_Min_Bat_1.na;
GVL.IOVD.X_U_Min_Bat_1.x					:= GVL.IIME.X_U_Min_Bat.x;
GVL.IOVD.X_U_Min_Bat_1.e					:= GVL.IIME.X_U_Min_Bat.e;
GVL.IOVD.X_U_Min_Bat_1.na					:= GVL.IIME.X_U_Min_Bat.na;
GVL.IOVD.X_U_Min_Bat_1.RangeExcd			:= (850 < GVL.IOVD.X_U_Min_Bat_1.x) OR (0 > GVL.IOVD.X_U_Min_Bat_1.x);
//-------SIGNAL -> X_U_Min_Cell_2 Max: 4 Min: 0 Def: 0 Resolution: 0.01 Offset: 0
GVL.IOVD.X_U_Min_Bat_2.v					:= GVL.SY.S_ECU_Rdy AND NOT GVL.IOVD.X_U_Min_Bat_2.e AND NOT GVL.IOVD.X_U_Min_Bat_2.na;
GVL.IOVD.X_U_Min_Bat_2.x					:= GVL.IIME.X_U_Min_Bat.x;
GVL.IOVD.X_U_Min_Bat_2.e					:= GVL.IIME.X_U_Min_Bat.e;
GVL.IOVD.X_U_Min_Bat_2.na					:= GVL.IIME.X_U_Min_Bat.na;
GVL.IOVD.X_U_Min_Bat_2.RangeExcd			:= (850 < GVL.IOVD.X_U_Min_Bat_2.x) OR (0 > GVL.IOVD.X_U_Min_Bat_2.x);
//-------SIGNAL -> X_U_Min_Cell_3 Max: 4 Min: 0 Def: 0 Resolution: 0.01 Offset: 0
GVL.IOVD.X_U_Min_Bat_3.v					:= GVL.SY.S_ECU_Rdy AND NOT GVL.IOVD.X_U_Min_Bat_3.e AND NOT GVL.IOVD.X_U_Min_Bat_3.na;
GVL.IOVD.X_U_Min_Bat_3.x					:= GVL.IIME.X_U_Min_Bat.x;
GVL.IOVD.X_U_Min_Bat_3.e					:= GVL.IIME.X_U_Min_Bat.e;
GVL.IOVD.X_U_Min_Bat_3.na					:= GVL.IIME.X_U_Min_Bat.na;
GVL.IOVD.X_U_Min_Bat_3.RangeExcd			:= (850 < GVL.IOVD.X_U_Min_Bat_3.x) OR (0 > GVL.IOVD.X_U_Min_Bat_3.x);
//-------SIGNAL -> X_U_Min_Cell_4 Max: 4 Min: 0 Def: 0 Resolution: 0.01 Offset: 0
GVL.IOVD.X_U_Min_Bat_4.v					:= GVL.SY.S_ECU_Rdy AND NOT GVL.IOVD.X_U_Min_Bat_4.e AND NOT GVL.IOVD.X_U_Min_Bat_4.na;
GVL.IOVD.X_U_Min_Bat_4.x					:= GVL.IIME.X_U_Min_Bat.x;
GVL.IOVD.X_U_Min_Bat_4.e					:= GVL.IIME.X_U_Min_Bat.e;
GVL.IOVD.X_U_Min_Bat_4.na					:= GVL.IIME.X_U_Min_Bat.na;
GVL.IOVD.X_U_Min_Bat_4.RangeExcd			:= (850 < GVL.IOVD.X_U_Min_Bat_4.x) OR (0 > GVL.IOVD.X_U_Min_Bat_4.x);
{endregion}
//-----------------------------------------------------------------------------------------------------------------------------
//-----------------------------------------------------------------------------------------------------------------------------
//MESSAGE------
{region " User Area : ESS_Ortalama_Hucre_Voltaji- ID:435"}

//-------SIGNAL -> X_U_Avg_Cell_1 Max: 4 Min: 0 Def: 0 Resolution: 0.01 Offset: 0
GVL.IOVD.X_U_Avg_Cell_1.v					:= GVL.SY.S_ECU_Rdy AND NOT GVL.IOVD.X_U_Avg_Cell_1.e AND NOT GVL.IOVD.X_U_Avg_Cell_1.na;
GVL.IOVD.X_U_Avg_Cell_1.x					:= GVL.ME.X_U_Avg_Bat;
GVL.IOVD.X_U_Avg_Cell_1.e					:= GVL.IIME.X_U_Min_Bat.e OR GVL.IIME.X_U_Max_Act_Bat.e;
GVL.IOVD.X_U_Avg_Cell_1.na					:= GVL.IIME.X_U_Min_Bat.na OR GVL.IIME.X_U_Max_Act_Bat.na;
GVL.IOVD.X_U_Avg_Cell_1.RangeExcd			:= (4 < GVL.IOVD.X_U_Avg_Cell_1.x) OR (0 > GVL.IOVD.X_U_Avg_Cell_1.x);
//-------SIGNAL -> X_U_Avg_Cell_2 Max: 4 Min: 0 Def: 0 Resolution: 0.01 Offset: 0
GVL.IOVD.X_U_Avg_Cell_2.v					:= GVL.SY.S_ECU_Rdy AND NOT GVL.IOVD.X_U_Avg_Cell_2.e AND NOT GVL.IOVD.X_U_Avg_Cell_2.na;
GVL.IOVD.X_U_Avg_Cell_2.x					:= GVL.ME.X_U_Avg_Bat;
GVL.IOVD.X_U_Avg_Cell_2.e					:= GVL.IIME.X_U_Min_Bat.e OR GVL.IIME.X_U_Max_Act_Bat.e;
GVL.IOVD.X_U_Avg_Cell_2.na					:= GVL.IIME.X_U_Min_Bat.na OR GVL.IIME.X_U_Max_Act_Bat.na;
GVL.IOVD.X_U_Avg_Cell_2.RangeExcd			:= (4 < GVL.IOVD.X_U_Avg_Cell_2.x) OR (0 > GVL.IOVD.X_U_Avg_Cell_2.x);
//-------SIGNAL -> X_U_Avg_Cell_3 Max: 4 Min: 0 Def: 0 Resolution: 0.01 Offset: 0
GVL.IOVD.X_U_Avg_Cell_3.v					:= GVL.SY.S_ECU_Rdy AND NOT GVL.IOVD.X_U_Avg_Cell_3.e AND NOT GVL.IOVD.X_U_Avg_Cell_3.na;
GVL.IOVD.X_U_Avg_Cell_3.x					:= GVL.ME.X_U_Avg_Bat;
GVL.IOVD.X_U_Avg_Cell_3.e					:= GVL.IIME.X_U_Min_Bat.e OR GVL.IIME.X_U_Max_Act_Bat.e;
GVL.IOVD.X_U_Avg_Cell_3.na					:= GVL.IIME.X_U_Min_Bat.na OR GVL.IIME.X_U_Max_Act_Bat.na;
GVL.IOVD.X_U_Avg_Cell_3.RangeExcd			:= (4 < GVL.IOVD.X_U_Avg_Cell_3.x) OR (0 > GVL.IOVD.X_U_Avg_Cell_3.x);
//-------SIGNAL -> X_U_Avg_Cell_4 Max: 4 Min: 0 Def: 0 Resolution: 0.01 Offset: 0
GVL.IOVD.X_U_Avg_Cell_4.v					:= GVL.SY.S_ECU_Rdy AND NOT GVL.IOVD.X_U_Avg_Cell_4.e AND NOT GVL.IOVD.X_U_Avg_Cell_4.na;
GVL.IOVD.X_U_Avg_Cell_4.x					:= 0;
GVL.IOVD.X_U_Avg_Cell_4.e					:= FALSE;
GVL.IOVD.X_U_Avg_Cell_4.na					:= FALSE;
GVL.IOVD.X_U_Avg_Cell_4.RangeExcd			:= (4 < GVL.IOVD.X_U_Avg_Cell_4.x) OR (0 > GVL.IOVD.X_U_Avg_Cell_4.x);
{endregion}
//-----------------------------------------------------------------------------------------------------------------------------
//-----------------------------------------------------------------------------------------------------------------------------
//MESSAGE------
{region " User Area : ESS_Sicaklik- ID:436"}

//-------SIGNAL -> X_T_Max_Cell_1 Max: 150 Min: -40 Def: 0 Resolution: 1 Offset: -40
GVL.IOVD.X_T_Max_Bat_1.v					:= GVL.SY.S_ECU_Rdy AND NOT GVL.IOVD.X_T_Max_Bat_1.e AND NOT GVL.IOVD.X_T_Max_Bat_1.na AND NOT GVL.IOVD.X_T_Max_Bat_1.RangeExcd;
GVL.IOVD.X_T_Max_Bat_1.x					:= GVL.IIME.X_T_Max_Bat.x;
GVL.IOVD.X_T_Max_Bat_1.e					:= GVL.IIME.X_T_Max_Bat.e;
GVL.IOVD.X_T_Max_Bat_1.na					:= GVL.IIME.X_T_Max_Bat.na;
GVL.IOVD.X_T_Max_Bat_1.RangeExcd			:= (150 < GVL.IOVD.X_T_Max_Bat_1.x) OR (-40 > GVL.IOVD.X_T_Max_Bat_1.x);
//-------SIGNAL -> X_T_Max_Cell_2 Max: 150 Min: -40 Def: 0 Resolution: 1 Offset: -40
GVL.IOVD.X_T_Max_Bat_2.v					:= GVL.SY.S_ECU_Rdy AND NOT GVL.IOVD.X_T_Max_Bat_2.e AND NOT GVL.IOVD.X_T_Max_Bat_2.na AND NOT GVL.IOVD.X_T_Max_Bat_2.RangeExcd;
GVL.IOVD.X_T_Max_Bat_2.x					:= GVL.IIME.X_T_Max_Bat.x; 
GVL.IOVD.X_T_Max_Bat_2.e					:= GVL.IIME.X_T_Max_Bat.e; 
GVL.IOVD.X_T_Max_Bat_2.na					:= GVL.IIME.X_T_Max_Bat.na;
GVL.IOVD.X_T_Max_Bat_2.RangeExcd			:= (150 < GVL.IOVD.X_T_Max_Bat_2.x) OR (-40 > GVL.IOVD.X_T_Max_Bat_2.x);
//-------SIGNAL -> X_T_Max_Cell_3 Max: 150 Min: -40 Def: 0 Resolution: 1 Offset: -40
GVL.IOVD.X_T_Max_Bat_3.v					:= GVL.SY.S_ECU_Rdy AND NOT GVL.IOVD.X_T_Max_Bat_3.e AND NOT GVL.IOVD.X_T_Max_Bat_3.na AND NOT GVL.IOVD.X_T_Max_Bat_3.RangeExcd;
GVL.IOVD.X_T_Max_Bat_3.x					:= GVL.IIME.X_T_Max_Bat.x; 
GVL.IOVD.X_T_Max_Bat_3.e					:= GVL.IIME.X_T_Max_Bat.e; 
GVL.IOVD.X_T_Max_Bat_3.na					:= GVL.IIME.X_T_Max_Bat.na;
GVL.IOVD.X_T_Max_Bat_3.RangeExcd			:= (150 < GVL.IOVD.X_T_Max_Bat_3.x) OR (-40 > GVL.IOVD.X_T_Max_Bat_3.x);
//-------SIGNAL -> X_T_Min_Cell_1 Max: 150 Min: -40 Def: 0 Resolution: 1 Offset: -40
GVL.IOVD.X_T_Min_Bat_1.v					:= GVL.SY.S_ECU_Rdy AND NOT GVL.IOVD.X_T_Min_Bat_1.e AND NOT GVL.IOVD.X_T_Min_Bat_1.na AND NOT GVL.IOVD.X_T_Min_Bat_1.RangeExcd;
GVL.IOVD.X_T_Min_Bat_1.x					:= GVL.IIME.X_T_Min_Bat.x; 
GVL.IOVD.X_T_Min_Bat_1.e					:= GVL.IIME.X_T_Min_Bat.e; 
GVL.IOVD.X_T_Min_Bat_1.na					:= GVL.IIME.X_T_Min_Bat.na;
GVL.IOVD.X_T_Min_Bat_1.RangeExcd			:= (150 < GVL.IOVD.X_T_Min_Bat_1.x) OR (-40 > GVL.IOVD.X_T_Min_Bat_1.x);
//-------SIGNAL -> X_T_Min_Cell_2 Max: 150 Min: -40 Def: 0 Resolution: 1 Offset: -40
GVL.IOVD.X_T_Min_Bat_2.v					:= GVL.SY.S_ECU_Rdy AND NOT GVL.IOVD.X_T_Min_Bat_2.e AND NOT GVL.IOVD.X_T_Min_Bat_2.na AND NOT GVL.IOVD.X_T_Min_Bat_2.RangeExcd;
GVL.IOVD.X_T_Min_Bat_2.x					:= GVL.IIME.X_T_Min_Bat.x;
GVL.IOVD.X_T_Min_Bat_2.e					:= GVL.IIME.X_T_Min_Bat.e; 
GVL.IOVD.X_T_Min_Bat_2.na					:= GVL.IIME.X_T_Min_Bat.na;
GVL.IOVD.X_T_Min_Bat_2.RangeExcd			:= (150 < GVL.IOVD.X_T_Min_Bat_2.x) OR (-40 > GVL.IOVD.X_T_Min_Bat_2.x);
//-------SIGNAL -> X_T_Min_Cell_3 Max: 150 Min: -40 Def: 0 Resolution: 1 Offset: -40
// GVL.IOVD.X_T_Min_Bat_3.v					:= GVL.SY.S_ECU_Rdy AND NOT GVL.IOVD.X_T_Min_Bat_3.e AND NOT GVL.IOVD.X_T_Min_Bat_3.na AND NOT GVL.IOVD.X_T_Min_Bat_3.RangeExcd;
// GVL.IOVD.X_T_Min_Bat_3.x					:= GVL.IIMEP.X_T_Cell_Pac_3.x; 
// GVL.IOVD.X_T_Min_Bat_3.e					:= GVL.IIMEP.X_T_Cell_Pac_3.e; 
// GVL.IOVD.X_T_Min_Bat_3.na					:= GVL.IIMEP.X_T_Cell_Pac_3.na;
// GVL.IOVD.X_T_Min_Bat_3.RangeExcd			:= (150 < GVL.IOVD.X_T_Min_Bat_3.x) OR (-40 > GVL.IOVD.X_T_Min_Bat_3.x);
//-------SIGNAL -> X_T_Avg_Bat_1 Max: 150 Min: -40 Def: 0 Resolution: 1 Offset: -40
GVL.IOVD.X_T_Avg_Bat_1.v					:= GVL.SY.S_ECU_Rdy AND NOT GVL.IOVD.X_T_Avg_Bat_1.e AND NOT GVL.IOVD.X_T_Avg_Bat_1.na AND NOT GVL.IOVD.X_T_Avg_Bat_1.RangeExcd;
GVL.IOVD.X_T_Avg_Bat_1.x					:= GVL.ME.X_T_Avg_Bat;    
GVL.IOVD.X_T_Avg_Bat_1.e					:= GVL.IIME.X_T_Max_Bat.e OR GVL.IIME.X_T_Min_Bat.e;
GVL.IOVD.X_T_Avg_Bat_1.na					:= GVL.IIME.X_T_Max_Bat.na OR GVL.IIME.X_T_Min_Bat.na;
GVL.IOVD.X_T_Avg_Bat_1.RangeExcd			:= (150 < GVL.IOVD.X_T_Avg_Bat_1.x) OR (-40 > GVL.IOVD.X_T_Avg_Bat_1.x);
{endregion}
//-----------------------------------------------------------------------------------------------------------------------------
//-----------------------------------------------------------------------------------------------------------------------------
//MESSAGE------
{region " User Area : ESS_Analog- ID:437"}

//-------SIGNAL -> X_I_Max_Chrg Max: 3000 Min: -3000 Def: 0 Resolution: 0.1 Offset: -3000
GVL.IOVD.X_I_Max_Chrg.v					:= GVL.SY.S_ECU_Rdy AND NOT GVL.IOVD.X_I_Max_Chrg.e AND NOT GVL.IOVD.X_I_Max_Chrg.na;
GVL.IOVD.X_I_Max_Chrg.x					:= GVL.IIME.X_I_Max_Act_Chrg.x;
GVL.IOVD.X_I_Max_Chrg.e					:= GVL.IIME.X_I_Max_Act_Chrg.e;
GVL.IOVD.X_I_Max_Chrg.na				:= GVL.IIME.X_I_Max_Act_Chrg.na;
GVL.IOVD.X_I_Max_Chrg.RangeExcd			:= (3000 < GVL.IOVD.X_I_Max_Chrg.x) OR (-3000 > GVL.IOVD.X_I_Max_Chrg.x);
//-------SIGNAL -> X_I_Max_Dischrg Max: 3000 Min: -3000 Def: 0 Resolution: 0.1 Offset: -3000
GVL.IOVD.X_I_Max_Dischrg.v				:= GVL.SY.S_ECU_Rdy AND NOT GVL.IOVD.X_I_Max_Dischrg.e AND NOT GVL.IOVD.X_I_Max_Dischrg.na;
GVL.IOVD.X_I_Max_Dischrg.x				:= GVL.IIME.X_I_Max_Act_DisChrg.x;
GVL.IOVD.X_I_Max_Dischrg.e				:= GVL.IIME.X_I_Max_Act_DisChrg.e;
GVL.IOVD.X_I_Max_Dischrg.na				:= GVL.IIME.X_I_Max_Act_DisChrg.na;
GVL.IOVD.X_I_Max_Dischrg.RangeExcd		:= (3000 < GVL.IOVD.X_I_Max_Dischrg.x) OR (-3000 > GVL.IOVD.X_I_Max_Dischrg.x);
//-------SIGNAL -> X_U_Tot_Bat Max: 1000 Min: 0 Def: 0 Resolution: 0.1 Offset: 0
GVL.IOVD.X_U_Tot_Bat.v					:= GVL.SY.S_ECU_Rdy AND NOT GVL.IOVD.X_U_Tot_Bat.e AND NOT GVL.IOVD.X_U_Tot_Bat.na;
GVL.IOVD.X_U_Tot_Bat.x					:= GVL.IIME.X_U_Act_Bat.x; 
GVL.IOVD.X_U_Tot_Bat.e					:= GVL.IIME.X_U_Act_Bat.e;
GVL.IOVD.X_U_Tot_Bat.na					:= GVL.IIME.X_U_Act_Bat.na;
GVL.IOVD.X_U_Tot_Bat.RangeExcd			:= (1000 < GVL.IOVD.X_U_Tot_Bat.x) OR (0 > GVL.IOVD.X_U_Tot_Bat.x);
{endregion}
//-----------------------------------------------------------------------------------------------------------------------------
//-----------------------------------------------------------------------------------------------------------------------------
//MESSAGE------
{region " User Area : ESS_Sogutma_Suyu- ID:438"}

//-------SIGNAL -> W_T_Clt Max: 200 Min: -40 Def: 0 Resolution: 1 Offset: -40
GVL.IOVD.W_T_Clt.v					:= GVL.SY.S_ECU_Rdy AND NOT GVL.IOVD.W_T_Clt.e AND NOT GVL.IOVD.W_T_Clt.na AND NOT GVL.IOVD.W_T_Clt.RangeExcd;
GVL.IOVD.W_T_Clt.x					:= 0;
GVL.IOVD.W_T_Clt.e					:= FALSE;
GVL.IOVD.W_T_Clt.na					:= FALSE;
GVL.IOVD.W_T_Clt.RangeExcd			:= (200 < GVL.IOVD.W_T_Clt.x) OR (-40 > GVL.IOVD.W_T_Clt.x);
//-------SIGNAL -> X_T_Clt Max: 200 Min: -40 Def: 0 Resolution: 1 Offset: -40
GVL.IOVD.X_T_Clt.v					:= GVL.SY.S_ECU_Rdy AND NOT GVL.IOVD.X_T_Clt.e AND NOT GVL.IOVD.X_T_Clt.na AND NOT GVL.IOVD.X_T_Clt.RangeExcd;
GVL.IOVD.X_T_Clt.x					:= 0;    
GVL.IOVD.X_T_Clt.e					:= FALSE;
GVL.IOVD.X_T_Clt.na					:= FALSE;
GVL.IOVD.X_T_Clt.RangeExcd			:= (200 < GVL.IOVD.X_T_Clt.x) OR (-40 > GVL.IOVD.X_T_Clt.x);
{endregion}
//-----------------------------------------------------------------------------------------------------------------------------
//-----------------------------------------------------------------------------------------------------------------------------
//MESSAGE------
{region " User Area : Sarj_Durum- ID:4A0"}

//-------SIGNAL -> S_Vh_Chrg_Perm Max: 1 Min: 0 Def: 0 Resolution: 1 Offset: 0
GVL.IOVD.S_Vh_Chrg_Perm.v					:= GVL.SY.S_ECU_Rdy AND NOT GVL.IOVD.S_Vh_Chrg_Perm.e AND NOT GVL.IOVD.S_Vh_Chrg_Perm.na;
GVL.IOVD.S_Vh_Chrg_Perm.x					:= GVL.MC.C_Chrg_Req;
GVL.IOVD.S_Vh_Chrg_Perm.e					:= GVL.MC.S_Err_Chrg;
GVL.IOVD.S_Vh_Chrg_Perm.na					:= FALSE;
//-------SIGNAL -> S_Vh_Insu_Meas Max: 1 Min: 0 Def: 0 Resolution: 1 Offset: 0
GVL.IOVD.S_Vh_Insu_Meas.v					:= GVL.SY.S_ECU_Rdy AND NOT GVL.IOVD.S_Vh_Insu_Meas.e AND NOT GVL.IOVD.S_Vh_Insu_Meas.na;
GVL.IOVD.S_Vh_Insu_Meas.x					:= GVL.IOPT.C_UKSI_MAN_TST_RQ.x OR GVL.IOPT.C_Insu_Tst_Req.x;
GVL.IOVD.S_Vh_Insu_Meas.e					:= GVL.IOPT.C_UKSI_MAN_TST_RQ.e OR GVL.IOPT.C_Insu_Tst_Req.e;
GVL.IOVD.S_Vh_Insu_Meas.na					:= GVL.IOPT.C_UKSI_MAN_TST_RQ.na OR GVL.IOPT.C_Insu_Tst_Req.na;
//-------SIGNAL -> S_Vh_Mobil Max: 1 Min: 0 Def: 0 Resolution: 1 Offset: 0
GVL.IOVD.S_Vh_Mobil.v						:= GVL.SY.S_ECU_Rdy AND NOT GVL.IOVD.S_Vh_Mobil.e AND NOT GVL.IOVD.S_Vh_Mobil.na;
GVL.IOVD.S_Vh_Mobil.x						:= 0;
GVL.IOVD.S_Vh_Mobil.e						:= FALSE;
GVL.IOVD.S_Vh_Mobil.na						:= FALSE;
//-------SIGNAL -> S_Chrg_Cmpl Max: 1 Min: 0 Def: 0 Resolution: 1 Offset: 0
GVL.IOVD.S_Chrg_Cmpl.v						:= GVL.SY.S_ECU_Rdy AND NOT GVL.IOVD.S_Chrg_Cmpl.e AND NOT GVL.IOVD.S_Chrg_Cmpl.na;
GVL.IOVD.S_Chrg_Cmpl.x						:= GVL.MC.S_Chrg_Fn;
GVL.IOVD.S_Chrg_Cmpl.e						:= GVL.MC.S_Err_Chrg;
GVL.IOVD.S_Chrg_Cmpl.na						:= FALSE;
//-------SIGNAL -> S_EV_Rdy Max: 1 Min: 0 Def: 0 Resolution: 1 Offset: 0
GVL.IOVD.S_EV_Rdy.v							:= GVL.SY.S_ECU_Rdy AND NOT GVL.IOVD.S_EV_Rdy.e AND NOT GVL.IOVD.S_EV_Rdy.na;
GVL.IOVD.S_EV_Rdy.x							:= GVL.MC.C_Chrg_Req;
GVL.IOVD.S_EV_Rdy.e							:= GVL.MC.S_Err_Chrg;
GVL.IOVD.S_EV_Rdy.na						:= FALSE;
//-------SIGNAL -> C_Chrg_Btn_Lft_Bwd_Led_Ctrl Max: 1 Min: 0 Def: 0 Resolution: 1 Offset: 0
GVL.IOVD.C_Chrg_Btn_Lft_Bwd_Led_Ctrl.v		:= GVL.SY.S_ECU_Rdy AND NOT GVL.IOVD.C_Chrg_Btn_Lft_Bwd_Led_Ctrl.e AND NOT GVL.IOVD.C_Chrg_Btn_Lft_Bwd_Led_Ctrl.na;
GVL.IOVD.C_Chrg_Btn_Lft_Bwd_Led_Ctrl.x		:= GVL.MC.C_Chrg_Btn_Lft_Bwd_Led_Ctrl;
GVL.IOVD.C_Chrg_Btn_Lft_Bwd_Led_Ctrl.e		:= FALSE;
GVL.IOVD.C_Chrg_Btn_Lft_Bwd_Led_Ctrl.na		:= FALSE;

//-------SIGNAL -> S_Pnt_Chrg_Mode_Sel Max: 1 Min: 0 Def: 0 Resolution: 1 Offset: 0
(*GVL.IOVD.S_Pnt_Chrg_Mode_Sel.v				:= GVL.SY.S_ECU_Rdy AND NOT GVL.IOVD.S_Pnt_Chrg_Mode_Sel.e AND NOT GVL.IOVD.S_Pnt_Chrg_Mode_Sel.na;
GVL.IOVD.S_Pnt_Chrg_Mode_Sel.x				:= ASSIGN HERE VALIDITY VARIABLE !!;
GVL.IOVD.S_Pnt_Chrg_Mode_Sel.e				:= ASSIGN HERE ERROR FLAG VARIABLE !!;
GVL.IOVD.S_Pnt_Chrg_Mode_Sel.na				:= ASSIGN HERE NOT AVAILABLE FLAG VARIABLE !!;
//-------SIGNAL -> S_Pnt_Chrg_Mode Max: 1 Min: 0 Def: 0 Resolution: 1 Offset: 0
GVL.IOVD.S_Pnt_Chrg_Mode.v					:= GVL.SY.S_ECU_Rdy AND NOT GVL.IOVD.S_Pnt_Chrg_Mode.e AND NOT GVL.IOVD.S_Pnt_Chrg_Mode.na;
GVL.IOVD.S_Pnt_Chrg_Mode.x					:= ASSIGN HERE VALIDITY VARIABLE !!;
GVL.IOVD.S_Pnt_Chrg_Mode.e					:= ASSIGN HERE ERROR FLAG VARIABLE !!;
GVL.IOVD.S_Pnt_Chrg_Mode.na					:= ASSIGN HERE NOT AVAILABLE FLAG VARIABLE !!;
//-------SIGNAL -> S_TCU_Pnt_Chrg_Ct Max: 1 Min: 0 Def: 0 Resolution: 1 Offset: 0
GVL.IOVD.S_TCU_Pnt_Chrg_Ct.v				:= GVL.SY.S_ECU_Rdy AND NOT GVL.IOVD.S_TCU_Pnt_Chrg_Ct.e AND NOT GVL.IOVD.S_TCU_Pnt_Chrg_Ct.na;
GVL.IOVD.S_TCU_Pnt_Chrg_Ct.x				:= ASSIGN HERE VALIDITY VARIABLE !!;
GVL.IOVD.S_TCU_Pnt_Chrg_Ct.e				:= ASSIGN HERE ERROR FLAG VARIABLE !!;
GVL.IOVD.S_TCU_Pnt_Chrg_Ct.na				:= ASSIGN HERE NOT AVAILABLE FLAG VARIABLE !!;
*)
//-------SIGNAL -> S_TCU_Chrg_Ct Max: 1 Min: 0 Def: 0 Resolution: 1 Offset: 0
GVL.IOVD.S_TCU_Chrg_Ct.v					:= GVL.SY.S_ECU_Rdy AND NOT GVL.IOVD.S_TCU_Chrg_Ct.e AND NOT GVL.IOVD.S_TCU_Chrg_Ct.na;
GVL.IOVD.S_TCU_Chrg_Ct.x					:= FALSE;
GVL.IOVD.S_TCU_Chrg_Ct.e					:= FALSE; 
GVL.IOVD.S_TCU_Chrg_Ct.na					:= FALSE;
{endregion}
//-----------------------------------------------------------------------------------------------------------------------------
//-----------------------------------------------------------------------------------------------------------------------------
//MESSAGE------
{region " User Area : Sarj_Sureleri- ID:4A5"}

//-------SIGNAL -> X_Tm_Seri_Hour Max: 250 Min: 0 Def: 0 Resolution: 1 Offset: 0
GVL.IOVD.X_Tm_Seri_Hour.v						:= GVL.SY.S_ECU_Rdy AND NOT GVL.IOVD.X_Tm_Seri_Hour.e AND NOT GVL.IOVD.X_Tm_Seri_Hour.na AND NOT GVL.IOVD.X_Tm_Seri_Hour.RangeExcd;
GVL.IOVD.X_Tm_Seri_Hour.x						:= GVL.MC.X_Lft_Chrg_Tm_Hour;
GVL.IOVD.X_Tm_Seri_Hour.e						:= FALSE;
GVL.IOVD.X_Tm_Seri_Hour.na						:= FALSE;
GVL.IOVD.X_Tm_Seri_Hour.RangeExcd				:=  (250 < GVL.IOVD.X_Tm_Seri_Hour.x) OR (0 > GVL.IOVD.X_Tm_Seri_Hour.x);
//-------SIGNAL -> X_Tm_Seri_Minute Max: 59 Min: 0 Def: 0 Resolution: 1 Offset: 0
GVL.IOVD.X_Tm_Seri_Minute.v						:= GVL.SY.S_ECU_Rdy AND NOT GVL.IOVD.X_Tm_Seri_Minute.e AND NOT GVL.IOVD.X_Tm_Seri_Minute.na AND NOT GVL.IOVD.X_Tm_Seri_Minute.RangeExcd;
GVL.IOVD.X_Tm_Seri_Minute.x						:= GVL.MC.X_Lft_Chrg_Tm_Min;
GVL.IOVD.X_Tm_Seri_Minute.e						:= FALSE;
GVL.IOVD.X_Tm_Seri_Minute.na					:= FALSE;
GVL.IOVD.X_Tm_Seri_Minute.RangeExcd				:=  (59 < GVL.IOVD.X_Tm_Seri_Minute.x) OR (0 > GVL.IOVD.X_Tm_Seri_Minute.x);
//-------SIGNAL -> X_Tm_Sp_Mode_Hour Max: 250 Min: 0 Def: 0 Resolution: 1 Offset: 0
GVL.IOVD.X_Tm_Sp_Mode_Hour.v					:= GVL.SY.S_ECU_Rdy AND NOT GVL.IOVD.X_Tm_Sp_Mode_Hour.e AND NOT GVL.IOVD.X_Tm_Sp_Mode_Hour.na AND NOT GVL.IOVD.X_Tm_Sp_Mode_Hour.RangeExcd;
GVL.IOVD.X_Tm_Sp_Mode_Hour.x					:= 0;
GVL.IOVD.X_Tm_Sp_Mode_Hour.e					:= FALSE;
GVL.IOVD.X_Tm_Sp_Mode_Hour.na					:= FALSE;
GVL.IOVD.X_Tm_Sp_Mode_Hour.RangeExcd			:=  (250 < GVL.IOVD.X_Tm_Sp_Mode_Hour.x) OR (0 > GVL.IOVD.X_Tm_Sp_Mode_Hour.x);
//-------SIGNAL -> X_Tm_Sp_Mode_Minute Max: 59 Min: 0 Def: 0 Resolution: 1 Offset: 0
GVL.IOVD.X_Tm_Sp_Mode_Minute.v					:= GVL.SY.S_ECU_Rdy AND NOT GVL.IOVD.X_Tm_Sp_Mode_Minute.e AND NOT GVL.IOVD.X_Tm_Sp_Mode_Minute.na AND NOT GVL.IOVD.X_Tm_Sp_Mode_Minute.RangeExcd;
GVL.IOVD.X_Tm_Sp_Mode_Minute.x					:= 0;
GVL.IOVD.X_Tm_Sp_Mode_Minute.e					:= FALSE;
GVL.IOVD.X_Tm_Sp_Mode_Minute.na					:= FALSE;
GVL.IOVD.X_Tm_Sp_Mode_Minute.RangeExcd			:=  (59 < GVL.IOVD.X_Tm_Sp_Mode_Minute.x) OR (0 > GVL.IOVD.X_Tm_Sp_Mode_Minute.x);
//-------SIGNAL -> X_Tm_Estm_Fn_Hour Max: 250 Min: 0 Def: 0 Resolution: 1 Offset: 0
GVL.IOVD.X_Tm_Estm_Fn_Hour.v					:= GVL.SY.S_ECU_Rdy AND NOT GVL.IOVD.X_Tm_Estm_Fn_Hour.e AND NOT GVL.IOVD.X_Tm_Estm_Fn_Hour.na AND NOT GVL.IOVD.X_Tm_Estm_Fn_Hour.RangeExcd;
GVL.IOVD.X_Tm_Estm_Fn_Hour.e					:= FALSE;
GVL.IOVD.X_Tm_Estm_Fn_Hour.na					:= FALSE;
GVL.IOVD.X_Tm_Estm_Fn_Hour.RangeExcd			:=  (250 < GVL.IOVD.X_Tm_Estm_Fn_Hour.x) OR (0 > GVL.IOVD.X_Tm_Estm_Fn_Hour.x);
//-------SIGNAL -> X_Tm_Estm_Fn_Minute Max: 59 Min: 0 Def: 0 Resolution: 1 Offset: 0
GVL.IOVD.X_Tm_Estm_Fn_Minute.v					:= GVL.SY.S_ECU_Rdy AND NOT GVL.IOVD.X_Tm_Estm_Fn_Minute.e AND NOT GVL.IOVD.X_Tm_Estm_Fn_Minute.na AND NOT GVL.IOVD.X_Tm_Estm_Fn_Minute.RangeExcd;
GVL.IOVD.X_Tm_Estm_Fn_Minute.e					:= FALSE;
GVL.IOVD.X_Tm_Estm_Fn_Minute.na					:= FALSE; 
GVL.IOVD.X_Tm_Estm_Fn_Minute.RangeExcd			:=  (59 < GVL.IOVD.X_Tm_Estm_Fn_Minute.x) OR (0 > GVL.IOVD.X_Tm_Estm_Fn_Minute.x);
{endregion}
//-----------------------------------------------------------------------------------------------------------------------------
//-----------------------------------------------------------------------------------------------------------------------------
//MESSAGE------
{region " User Area : Sarj_Durum_3- ID:4A6"}

//-------SIGNAL -> Z_Ext_Chrg_Stat Max: 255 Min: 0 Def: 0 Resolution: 1 Offset: 0
GVL.IOVD.Z_Ext_Chrg_Stat.v					:= GVL.SY.S_ECU_Rdy AND NOT GVL.IOVD.Z_Ext_Chrg_Stat.e AND NOT GVL.IOVD.Z_Ext_Chrg_Stat.na AND NOT GVL.IOVD.Z_Ext_Chrg_Stat.RangeExcd;
	
// PR1006_SRS_001099_TIMTRO
// PR1006_SRS_001102_TIMTRO
// PR1006_SRS_001100_TIMTRO
_FB_PACK_8BITS_TO_BYTE_0(	S_BIT_0 := 0,
							S_BIT_1	:= ,
							S_BIT_2 := ,
							S_BIT_3 := 0,
							S_BIT_4 := GVL.MC.S_Inlt_Conn,
							S_BIT_5 := GVL.MC.S_Chrg_Req,
							S_BIT_6 := GVL.MC.S_Chrg_Actv,
							S_BIT_7 := GVL.MC.S_Err_Chrg,
							X_BYTE_0 => GVL.IOVD.Z_Ext_Chrg_Stat.x);
GVL.IOVD.Z_Ext_Chrg_Stat.e					:= FALSE;
GVL.IOVD.Z_Ext_Chrg_Stat.na					:= FALSE;
GVL.IOVD.Z_Ext_Chrg_Stat.RangeExcd			:=  (255 < GVL.IOVD.Z_Ext_Chrg_Stat.x) OR (0 > GVL.IOVD.Z_Ext_Chrg_Stat.x);
	 
// PR1006_REV_002449_TIMTRO
//-------SIGNAL -> Z_Pan_Chrg_Stat Max: 255 Min: 0 Def: 0 Resolution: 1 Offset: 0
_FB_PACK_8BITS_TO_BYTE_0(	S_BIT_0 := 0,													// Pantograph fast charger linked
							S_BIT_1	:= 0,													// Pantograf fast charge getting started
							S_BIT_2 := 0,													// Pantograph fast charge is active
							S_BIT_3 := 0,													// Pantograph fast charge fault
							S_BIT_4 := GVL.MP.S_Pnt_Chrg_Actv AND GVL.MP.S_Pol_Up,			// Catenary charge is getting started
							S_BIT_5 := GVL.MP.S_Pnt_Chrg_Actv AND GVL.MP.S_Pol_Up,			// Catenary charge is active
							S_BIT_6 := GVL.MP.S_Pnt_Chrg_Actv AND GVL.MP.S_Pol_Up AND GVL.ED_Typ.Tr_Ctrl[ED_Tr_Ctrl_E.S_Pnt_Chrg_Ct_Plus_Err].S_Evnt_Actv,	// Catenary charge fault
							S_BIT_7 := 0, // Spare
							X_BYTE_0 => GVL.IOVD.Z_Pan_Chrg_Stat.x);
GVL.IOVD.Z_Pan_Chrg_Stat.v					:= GVL.SY.S_ECU_Rdy AND NOT GVL.IOVD.Z_Pan_Chrg_Stat.e AND NOT GVL.IOVD.X_Tm_Estm_Fn_Minute.na AND NOT GVL.IOVD.Z_Pan_Chrg_Stat.RangeExcd;
GVL.IOVD.Z_Pan_Chrg_Stat.e					:= FALSE;
GVL.IOVD.Z_Pan_Chrg_Stat.na					:= FALSE;
GVL.IOVD.Z_Pan_Chrg_Stat.RangeExcd			:=  (255 < GVL.IOVD.Z_Pan_Chrg_Stat.x) OR (0 > GVL.IOVD.Z_Pan_Chrg_Stat.x);
//-------SIGNAL -> Z_Pnt_Pos Max: 255 Min: 0 Def: 0 Resolution: 1 Offset: 0
GVL.IOVD.Z_Pnt_Pos.v						:= GVL.SY.S_ECU_Rdy AND NOT GVL.IOVD.Z_Pnt_Pos.e AND NOT GVL.IOVD.Z_Pnt_Pos.na AND NOT GVL.IOVD.Z_Pnt_Pos.RangeExcd;
// GVL.IOVD.Z_Pnt_Pos.x						:= UINT_TO_BYTE (REAL_TO_UINT(GVL.IIMP.X_Poles_Stat.x));   
GVL.IOVD.Z_Pnt_Pos.e						:= FALSE;
GVL.IOVD.Z_Pnt_Pos.na						:= FALSE;
GVL.IOVD.Z_Pnt_Pos.RangeExcd				:=  (255 < GVL.IOVD.Z_Pnt_Pos.x) OR (0 > GVL.IOVD.Z_Pnt_Pos.x);
{endregion}
//-----------------------------------------------------------------------------------------------------------------------------
//-----------------------------------------------------------------------------------------------------------------------------
//MESSAGE------
// PR1006_REV_002449_TIMTRO
{region " User Area : Pantograph_Analog_4- ID:4AF"}
//-------SIGNAL -> X_I_Pnt_Chrg Max: 30000 Min: -32767 Def: 0 Resolution: 1 Offset: -32767
GVL.IOVD.X_I_Pnt_Chrg.v					:= GVL.SY.S_ECU_Rdy AND GVL.MP.S_Pnt_Chrg_Actv AND NOT GVL.IOVD.X_I_Pnt_Chrg.e AND NOT GVL.IOVD.X_I_Pnt_Chrg.na AND NOT GVL.IOVD.X_I_Pnt_Chrg.RangeExcd;
GVL.IOVD.X_I_Pnt_Chrg.x					:= GVL.IIME.X_I_Act_Bat.x;
GVL.IOVD.X_I_Pnt_Chrg.e					:= GVL.IIME.X_I_Act_Bat.e;
GVL.IOVD.X_I_Pnt_Chrg.na				:= GVL.IIME.X_I_Act_Bat.na;
GVL.IOVD.X_I_Pnt_Chrg.RangeExcd			:= (800 < GVL.IOVD.X_I_Pnt_Chrg.x) OR (-800 > GVL.IOVD.X_I_Pnt_Chrg.x);

//-------SIGNAL -> X_U_Pnt_Chrg Max: 30000 Min: -32767 Def: 0 Resolution: 1 Offset: -32767
GVL.IOVD.X_U_Pnt_Chrg.v					:= GVL.SY.S_ECU_Rdy AND GVL.MP.S_Pnt_Chrg_Actv AND NOT GVL.IOVD.X_U_Pnt_Chrg.e AND NOT GVL.IOVD.X_U_Pnt_Chrg.na AND NOT GVL.IOVD.X_U_Pnt_Chrg.RangeExcd;
GVL.IOVD.X_U_Pnt_Chrg.x					:= GVL.IIPT.X_U_DCDC_Out.x;
GVL.IOVD.X_U_Pnt_Chrg.e					:= GVL.IIPT.X_U_DCDC_Out.e;
GVL.IOVD.X_U_Pnt_Chrg.na				:= GVL.IIPT.X_U_DCDC_Out.na;
GVL.IOVD.X_U_Pnt_Chrg.RangeExcd			:= (1600 < GVL.IOVD.X_U_Pnt_Chrg.x) OR (0 > GVL.IOVD.X_U_Pnt_Chrg.x);

//-------SIGNAL X_P_Pnt_Chrg X_P_Pnt_Chrg Max: 3276 Min: -3276 Def: 0 Resolution: 0.1 Offset: 0
GVL.IOVD.X_P_Pnt_Chrg.v					:= GVL.SY.S_ECU_Rdy AND GVL.MP.S_Pnt_Chrg_Actv AND NOT GVL.IOVD.X_P_Pnt_Chrg.e AND NOT GVL.IOVD.X_P_Pnt_Chrg.na AND NOT GVL.IOVD.X_P_Pnt_Chrg.RangeExcd;
GVL.IOVD.X_P_Pnt_Chrg.x					:= GVL.IIPT.X_P_Out_DCDC.x;
GVL.IOVD.X_P_Pnt_Chrg.e					:= GVL.IIPT.X_P_Out_DCDC.e;
GVL.IOVD.X_P_Pnt_Chrg.na				:= GVL.IIPT.X_P_Out_DCDC.na;
GVL.IOVD.X_P_Pnt_Chrg.RangeExcd			:= (3276 < GVL.IOVD.X_P_Pnt_Chrg.x) OR (-3276 > GVL.IOVD.X_P_Pnt_Chrg.x);

//-------SIGNAL -> X_T_Pnt_Chrg Max: 210 Min: -40 Def: 0 Resolution: 1 Offset: -40
GVL.IOVD.X_T_Pnt_Chrg.v					:= GVL.SY.S_ECU_Rdy AND GVL.MP.S_Pnt_Chrg_Actv AND NOT GVL.IOVD.X_T_Pnt_Chrg.e AND NOT GVL.IOVD.X_T_Pnt_Chrg.na AND NOT GVL.IOVD.X_T_Pnt_Chrg.RangeExcd;
GVL.IOVD.X_T_Pnt_Chrg.x					:= GVL.IIPT.X_T_DCDC_Cnv.x;
GVL.IOVD.X_T_Pnt_Chrg.e					:= GVL.IIPT.X_T_DCDC_Cnv.e;
GVL.IOVD.X_T_Pnt_Chrg.na				:= GVL.IIPT.X_T_DCDC_Cnv.na;
GVL.IOVD.X_T_Pnt_Chrg.RangeExcd			:= (210 < GVL.IIPT.X_T_DCDC_Cnv.x) OR (-40 > GVL.IIPT.X_T_DCDC_Cnv.x);

{endregion}
//-----------------------------------------------------------------------------------------------------------------------------
//-----------------------------------------------------------------------------------------------------------------------------
//MESSAGE------
{region " User Area : Hava_Kompresoru_Durum- ID:4F0"}

//-------SIGNAL -> C_Air_Cmp_On Max: 1 Min: 0 Def: 0 Resolution: 1 Offset: 0
GVL.IOVD.C_Air_Cmp_On.v					:= GVL.SY.S_ECU_Rdy AND NOT GVL.IOVD.C_Air_Cmp_On.e AND NOT GVL.IOVD.C_Air_Cmp_On.na;
GVL.IOVD.C_Air_Cmp_On.x					:= GVL.IORE.C_Air_Cmp_On;
GVL.IOVD.C_Air_Cmp_On.e					:= FALSE;
GVL.IOVD.C_Air_Cmp_On.na				:= FALSE;
//-------SIGNAL -> S_Air_Cmp_On Max: 1 Min: 0 Def: 0 Resolution: 1 Offset: 0
GVL.IOVD.S_Air_Cmp_On.v					:= GVL.SY.S_ECU_Rdy AND NOT GVL.IOVD.S_Air_Cmp_On.e AND NOT GVL.IOVD.S_Air_Cmp_On.na;
GVL.IOVD.S_Air_Cmp_On.x					:= NOT GVL.IIRE.S_Air_Cmp_Ct_Deactv.pin_value;
GVL.IOVD.S_Air_Cmp_On.e					:= NOT GVL.IIRE.S_Air_Cmp_Ct_Deactv.error = lib500_types.IO_ERRORTYPE.IO_E_OK;
GVL.IOVD.S_Air_Cmp_On.na				:= FALSE;
//-------SIGNAL -> S_ER_Air_Cmp Max: 1 Min: 0 Def: 0 Resolution: 1 Offset: 0
GVL.IOVD.S_ER_Air_Cmp.v					:= GVL.SY.S_ECU_Rdy AND NOT GVL.IOVD.S_ER_Air_Cmp.e AND NOT GVL.IOVD.S_ER_Air_Cmp.na;
GVL.IOVD.S_ER_Air_Cmp.x					:= (GVL.XC.S_Air_Cmp_Ct_Err OR GVL.XC.S_ER_Air_Cmp_Tmp); //EKLENECEK
GVL.IOVD.S_ER_Air_Cmp.e					:= FALSE;
GVL.IOVD.S_ER_Air_Cmp.na				:= FALSE;
//-------SIGNAL -> S_ER_Hi_Temp_Air_Cmp Max: 1 Min: 0 Def: 0 Resolution: 1 Offset: 0
GVL.IOVD.S_ER_Hi_Temp_Air_Cmp.v			:= GVL.SY.S_ECU_Rdy AND NOT GVL.IOVD.S_ER_Hi_Temp_Air_Cmp.e AND NOT GVL.IOVD.S_ER_Hi_Temp_Air_Cmp.na;
GVL.IOVD.S_ER_Hi_Temp_Air_Cmp.x			:= GVL.XC.S_ER_Air_Cmp_Tmp;
GVL.IOVD.S_ER_Hi_Temp_Air_Cmp.e			:= FALSE;
GVL.IOVD.S_ER_Hi_Temp_Air_Cmp.na		:= FALSE;
//-------SIGNAL -> S_ER_Psb_Air_Lek Max: 1 Min: 0 Def: 0 Resolution: 1 Offset: 0
GVL.IOVD.S_ER_Psb_Air_Lek.v			:= GVL.SY.S_ECU_Rdy AND NOT GVL.IOVD.S_ER_Psb_Air_Lek.e AND NOT GVL.IOVD.S_ER_Psb_Air_Lek.na;
GVL.IOVD.S_ER_Psb_Air_Lek.x			:= GVL.XC.S_Psb_Air_Lek;
GVL.IOVD.S_ER_Psb_Air_Lek.e			:= FALSE;
GVL.IOVD.S_ER_Psb_Air_Lek.na		:= FALSE;
{endregion}
//-----------------------------------------------------------------------------------------------------------------------------
//-----------------------------------------------------------------------------------------------------------------------------
{region " MESSAGE AREA :ESS_Durum- ID:430"}

{region " SIGNAL AREA : NAME->S_ESS_Mn_Ct LENGTH->2 STARTBIT :0"}
_FB_CanTx_Message_Unpack_430.S_Bit_0		:= (GVL.IOVD.S_ESS_Mn_Ct.x OR GVL.IOVD.S_ESS_Mn_Ct.na) AND NOT GVL.IOVD.S_ESS_Mn_Ct.e; 
_FB_CanTx_Message_Unpack_430.S_Bit_1		:= NOT GVL.IOVD.S_ESS_Mn_Ct.v OR GVL.IOVD.S_ESS_Mn_Ct.na OR GVL.IOVD.S_ESS_Mn_Ct.e; 
{endregion}

{region " SIGNAL AREA : NAME->S_Insu_Ok LENGTH->2 STARTBIT :4"}
_FB_CanTx_Message_Unpack_430.S_Bit_4		:= (GVL.IOVD.S_Insu_Ok.x OR GVL.IOVD.S_Insu_Ok.na) AND NOT GVL.IOVD.S_Insu_Ok.e; 
_FB_CanTx_Message_Unpack_430.S_Bit_5		:= NOT GVL.IOVD.S_Insu_Ok.v OR GVL.IOVD.S_Insu_Ok.na OR GVL.IOVD.S_Insu_Ok.e; 
{endregion}

{region " SIGNAL AREA : NAME->S_BMS_Sp LENGTH->2 STARTBIT :6"}
_FB_CanTx_Message_Unpack_430.S_Bit_6		:= (GVL.IOVD.S_BMS_Sp.x OR GVL.IOVD.S_BMS_Sp.na) AND NOT GVL.IOVD.S_BMS_Sp.e; 
_FB_CanTx_Message_Unpack_430.S_Bit_7		:= NOT GVL.IOVD.S_BMS_Sp.v OR GVL.IOVD.S_BMS_Sp.na OR GVL.IOVD.S_BMS_Sp.e; 
{endregion}

{region " SIGNAL AREA : NAME->S_Bat_Mode LENGTH->2 STARTBIT :8"}
_FB_CanTx_Message_Unpack_430.S_Bit_8		:= (GVL.IOVD.S_Bat_Mode.x OR GVL.IOVD.S_Bat_Mode.na) AND NOT GVL.IOVD.S_Bat_Mode.e; 
_FB_CanTx_Message_Unpack_430.S_Bit_9		:= NOT GVL.IOVD.S_Bat_Mode.v OR GVL.IOVD.S_Bat_Mode.na OR GVL.IOVD.S_Bat_Mode.e; 
{endregion}

{region " SIGNAL AREA : NAME->S_Ops_Mode LENGTH->2 STARTBIT :10"}
_FB_CanTx_Message_Unpack_430.S_Bit_10		:= (GVL.IOVD.S_Ops_Mode.x OR GVL.IOVD.S_Ops_Mode.na) AND NOT GVL.IOVD.S_Ops_Mode.e; 
_FB_CanTx_Message_Unpack_430.S_Bit_11		:= NOT GVL.IOVD.S_Ops_Mode.v OR GVL.IOVD.S_Ops_Mode.na OR GVL.IOVD.S_Ops_Mode.e; 
{endregion}

{region " SIGNAL AREA : NAME->C_Tr_Mode LENGTH->2 STARTBIT :12"}
_FB_CanTx_Message_Unpack_430.S_Bit_12		:= (GVL.IOVD.C_Tr_Mode.x OR GVL.IOVD.C_Tr_Mode.na) AND NOT GVL.IOVD.C_Tr_Mode.e; 
_FB_CanTx_Message_Unpack_430.S_Bit_13		:= NOT GVL.IOVD.C_Tr_Mode.v OR GVL.IOVD.C_Tr_Mode.na OR GVL.IOVD.C_Tr_Mode.e; 
{endregion}

{region " SIGNAL AREA : NAME->S_Pwr_Distr LENGTH->2 STARTBIT :16"}
_FB_CanTx_Message_Unpack_430.S_Bit_16		:= (GVL.IOVD.S_Pwr_Distr.x OR GVL.IOVD.S_Pwr_Distr.na) AND NOT GVL.IOVD.S_Pwr_Distr.e; 
_FB_CanTx_Message_Unpack_430.S_Bit_17		:= NOT GVL.IOVD.S_Pwr_Distr.v OR GVL.IOVD.S_Pwr_Distr.na OR GVL.IOVD.S_Pwr_Distr.e; 
{endregion}

{region " SIGNAL AREA : NAME->S_Ext_Sp_Req LENGTH->2 STARTBIT :24"}
_FB_CanTx_Message_Unpack_430.S_Bit_24		:= (GVL.IOVD.S_Ext_Sp_Req.x OR GVL.IOVD.S_Ext_Sp_Req.na) AND NOT GVL.IOVD.S_Ext_Sp_Req.e; 
_FB_CanTx_Message_Unpack_430.S_Bit_25		:= NOT GVL.IOVD.S_Ext_Sp_Req.v OR GVL.IOVD.S_Ext_Sp_Req.na OR GVL.IOVD.S_Ext_Sp_Req.e; 
{endregion}

{region " SIGNAL AREA : NAME->S_Vh_Mode_Req LENGTH->2 STARTBIT :26"}
_FB_CanTx_Message_Unpack_430.S_Bit_26		:= (GVL.IOVD.X_Vh_Mode_Req.x = 3 OR GVL.IOVD.X_Vh_Mode_Req.na) AND NOT GVL.IOVD.X_Vh_Mode_Req.e; 
_FB_CanTx_Message_Unpack_430.S_Bit_27		:= NOT GVL.IOVD.X_Vh_Mode_Req.v OR GVL.IOVD.X_Vh_Mode_Req.na OR GVL.IOVD.X_Vh_Mode_Req.e; 
{endregion}

{region " SIGNAL AREA : NAME->Z_MBMS_Mode LENGTH->8 STARTBIT :32"}
_FB_CanTx_Message_Unpack_430.X_Byte_4					:=
(*SELECT 1 : Is data valid and range is not exceed?*)	SEL((GVL.IOVD.Z_MBMS_Mode.v AND NOT GVL.IOVD.Z_MBMS_Mode.RangeExcd),
(*SELECT 2 : Is NOT AVAILABLE ?*)						SEL(GVL.IOVD.Z_MBMS_Mode.na,
(*SELECT 3 : Is ERROR active ?*)						SEL(GVL.IOVD.Z_MBMS_Mode.e,
(*DEFAULT VALUE assignment*)							0,
(*ERROR is active*)										16#E),
(*NOT AVAILABLE is active*)								16#F),
(*Transmission is VALID*)								GVL.IOVD.Z_MBMS_Mode.x);
{endregion}

{region " SIGNAL AREA : NAME->Z_Bat_Ops LENGTH->4 STARTBIT :40"}
_FB_UNPACK_BYTE_TO_8BITS_0 (	S_Bit_0 => _FB_CanTx_Message_Unpack_430.S_Bit_40,
								S_Bit_1 => _FB_CanTx_Message_Unpack_430.S_Bit_41,
								S_Bit_2 => _FB_CanTx_Message_Unpack_430.S_Bit_42,
								S_Bit_3 => _FB_CanTx_Message_Unpack_430.S_Bit_43 ,
								X_BYTE_0				:=
(*SELECT 1 : Is data valid and range is not exceed?*)	SEL((GVL.IOVD.Z_Bat_Ops.v AND NOT GVL.IOVD.Z_Bat_Ops.RangeExcd),
(*SELECT 2 : Is NOT AVAILABLE ?*)						SEL(GVL.IOVD.Z_Bat_Ops.na,
(*SELECT 3 : Is ERROR active ?*)						SEL(GVL.IOVD.Z_Bat_Ops.e,
(*DEFAULT VALUE assignment*)							0,
(*ERROR is active*)										16#E),
(*NOT AVAILABLE is active*)								16#F),
(*Transmission is VALID*)								GVL.IOVD.Z_Bat_Ops.x));
{endregion}

